  PROC DrawPart25()
    MoveL Offs(pOrigin,198.50,118.14,0.00),v40,z0,tPen\WObj:=wPaper;
    MoveL Offs(pOrigin,175.10,118.14,0.00),v40,z0,tPen\WObj:=wPaper;
    MoveL Offs(pOrigin,174.22,118.63,0.00),v40,z0,tPen\WObj:=wPaper;
    MoveL Offs(pOrigin,188.97,133.37,0.00),v40,fine,tPen\WObj:=wPaper;
    MoveL Offs(pOrigin,188.97,133.37,6.00),v60,z5,tPen\WObj:=wPaper;
    MoveL Offs(pOrigin,188.05,134.17,6.00),vTravel,z5,tPen\WObj:=wPaper;
    MoveL Offs(pOrigin,188.05,134.17,0.00),v60,z0,tPen\WObj:=wPaper;
    MoveL Offs(pOrigin,199.82,122.39,0.00),v40,z0,tPen\WObj:=wPaper;
    MoveL Offs(pOrigin,199.21,122.71,0.00),v40,z0,tPen\WObj:=wPaper;
    MoveL Offs(pOrigin,174.18,97.67,0.00),v40,z0,tPen\WObj:=wPaper;
    MoveL Offs(pOrigin,174.95,98.07,0.00),v40,z0,tPen\WObj:=wPaper;
    MoveL Offs(pOrigin,198.65,98.07,0.00),v40,z0,tPen\WObj:=wPaper;
    MoveL Offs(pOrigin,199.39,97.50,0.00),v40,z0,tPen\WObj:=wPaper;
    MoveL Offs(pOrigin,195.04,93.15,0.00),v40,z0,tPen\WObj:=wPaper;
    MoveL Offs(pOrigin,195.48,92.38,0.00),v40,z0,tPen\WObj:=wPaper;
    MoveL Offs(pOrigin,173.52,114.34,0.00),v40,z0,tPen\WObj:=wPaper;
    MoveL Offs(pOrigin,174.24,114.16,0.00),v40,z0,tPen\WObj:=wPaper;
    MoveL Offs(pOrigin,193.43,133.36,0.00),v40,z0,tPen\WObj:=wPaper;
    MoveL Offs(pOrigin,194.00,134.18,0.00),v40,z0,tPen\WObj:=wPaper;
    MoveL Offs(pOrigin,200.15,128.03,0.00),v40,z0,tPen\WObj:=wPaper;
    MoveL Offs(pOrigin,199.41,127.39,0.00),v40,z0,tPen\WObj:=wPaper;
    MoveL Offs(pOrigin,174.16,102.14,0.00),v40,z0,tPen\WObj:=wPaper;
    MoveL Offs(pOrigin,174.95,102.30,0.00),v40,z0,tPen\WObj:=wPaper;
    MoveL Offs(pOrigin,198.50,102.30,0.00),v40,z0,tPen\WObj:=wPaper;
    MoveL Offs(pOrigin,199.16,101.75,0.00),v40,z0,tPen\WObj:=wPaper;
    MoveL Offs(pOrigin,190.57,93.16,0.00),v40,z0,tPen\WObj:=wPaper;
    MoveL Offs(pOrigin,191.12,92.27,0.00),v40,z0,tPen\WObj:=wPaper;
    MoveL Offs(pOrigin,173.40,109.98,0.00),v40,z0,tPen\WObj:=wPaper;
    MoveL Offs(pOrigin,174.25,109.69,0.00),v40,z0,tPen\WObj:=wPaper;
    MoveL Offs(pOrigin,197.90,133.35,0.00),v40,z0,tPen\WObj:=wPaper;
    MoveL Offs(pOrigin,197.19,133.98,0.00),v40,z0,tPen\WObj:=wPaper;
    MoveL Offs(pOrigin,224.03,107.14,0.00),v40,z0,tPen\WObj:=wPaper;
    MoveL Offs(pOrigin,223.28,106.40,0.00),v40,z0,tPen\WObj:=wPaper;
    MoveL Offs(pOrigin,201.11,128.57,0.00),v40,z0,tPen\WObj:=wPaper;
    MoveL Offs(pOrigin,201.85,128.34,0.00),v40,z0,tPen\WObj:=wPaper;
    MoveL Offs(pOrigin,206.84,133.32,0.00),v40,z0,tPen\WObj:=wPaper;
    MoveL Offs(pOrigin,207.40,134.22,0.00),v40,z0,tPen\WObj:=wPaper;
    MoveL Offs(pOrigin,225.97,115.66,0.00),v40,z0,tPen\WObj:=wPaper;
    MoveL Offs(pOrigin,224.97,115.61,0.00),v40,z0,tPen\WObj:=wPaper;
    MoveL Offs(pOrigin,202.80,93.45,0.00),v40,z0,tPen\WObj:=wPaper;
    MoveL Offs(pOrigin,202.85,92.93,0.00),v40,z0,tPen\WObj:=wPaper;
    MoveL Offs(pOrigin,218.60,92.93,0.00),v40,z0,tPen\WObj:=wPaper;
    MoveL Offs(pOrigin,202.85,92.93,0.00),v40,z0,tPen\WObj:=wPaper;
    MoveL Offs(pOrigin,202.71,92.62,0.00),v40,z0,tPen\WObj:=wPaper;
    MoveL Offs(pOrigin,201.55,93.78,0.00),v40,z0,tPen\WObj:=wPaper;
    MoveL Offs(pOrigin,201.95,93.53,0.00),v40,z0,tPen\WObj:=wPaper;
    MoveL Offs(pOrigin,201.95,94.72,0.00),v40,z0,tPen\WObj:=wPaper;
    MoveL Offs(pOrigin,201.95,93.53,0.00),v40,z0,tPen\WObj:=wPaper;
    MoveL Offs(pOrigin,202.16,94.30,0.00),v40,z0,tPen\WObj:=wPaper;
    MoveL Offs(pOrigin,224.97,117.10,0.00),v40,z0,tPen\WObj:=wPaper;
    MoveL Offs(pOrigin,224.15,117.08,0.00),v40,z0,tPen\WObj:=wPaper;
    MoveL Offs(pOrigin,203.00,117.08,0.00),v40,z0,tPen\WObj:=wPaper;
    MoveL Offs(pOrigin,202.20,116.74,0.00),v40,z0,tPen\WObj:=wPaper;
    MoveL Offs(pOrigin,216.31,130.85,0.00),v40,z0,tPen\WObj:=wPaper;
    MoveL Offs(pOrigin,217.10,130.48,0.00),v40,z0,tPen\WObj:=wPaper;
    MoveL Offs(pOrigin,219.35,128.77,0.00),v40,z0,tPen\WObj:=wPaper;
    MoveL Offs(pOrigin,220.70,127.43,0.00),v40,z0,tPen\WObj:=wPaper;
    MoveL Offs(pOrigin,223.00,124.12,0.00),v40,z0,tPen\WObj:=wPaper;
    MoveL Offs(pOrigin,224.20,121.43,0.00),v40,z0,tPen\WObj:=wPaper;
    MoveL Offs(pOrigin,225.05,118.12,0.00),v40,z0,tPen\WObj:=wPaper;
    MoveL Offs(pOrigin,225.05,113.03,0.00),v40,z0,tPen\WObj:=wPaper;
    MoveL Offs(pOrigin,223.90,108.97,0.00),v40,z0,tPen\WObj:=wPaper;
    MoveL Offs(pOrigin,222.70,106.57,0.00),v40,z0,tPen\WObj:=wPaper;
    MoveL Offs(pOrigin,220.55,103.72,0.00),v40,z0,tPen\WObj:=wPaper;
    MoveL Offs(pOrigin,217.75,101.32,0.00),v40,z0,tPen\WObj:=wPaper;
    MoveL Offs(pOrigin,220.60,99.28,0.00),v40,z0,tPen\WObj:=wPaper;
    MoveL Offs(pOrigin,201.95,106.28,0.00),v40,z0,tPen\WObj:=wPaper;
    MoveL Offs(pOrigin,202.00,133.07,0.00),v40,z0,tPen\WObj:=wPaper;
    MoveL Offs(pOrigin,208.55,133.27,0.00),v40,z0,tPen\WObj:=wPaper;
    MoveL Offs(pOrigin,213.80,132.12,0.00),v40,z0,tPen\WObj:=wPaper;
    MoveL Offs(pOrigin,217.10,130.48,0.00),v40,z0,tPen\WObj:=wPaper;
    MoveL Offs(pOrigin,217.27,130.31,0.00),v40,z0,tPen\WObj:=wPaper;
    MoveL Offs(pOrigin,202.21,115.25,0.00),v40,z0,tPen\WObj:=wPaper;
    MoveL Offs(pOrigin,201.50,114.74,0.00),v40,z0,tPen\WObj:=wPaper;
    MoveL Offs(pOrigin,224.20,92.04,0.00),v40,z0,tPen\WObj:=wPaper;
    MoveL Offs(pOrigin,224.71,92.96,0.00),v40,z0,tPen\WObj:=wPaper;
    MoveL Offs(pOrigin,226.20,94.44,0.00),v40,z0,tPen\WObj:=wPaper;
    MoveL Offs(pOrigin,225.45,95.19,0.00),v40,z0,tPen\WObj:=wPaper;
    MoveL Offs(pOrigin,223.23,92.96,0.00),v40,z0,tPen\WObj:=wPaper;
    MoveL Offs(pOrigin,222.71,92.04,0.00),v40,z0,tPen\WObj:=wPaper;
    MoveL Offs(pOrigin,201.49,113.25,0.00),v40,z0,tPen\WObj:=wPaper;
    MoveL Offs(pOrigin,202.21,113.76,0.00),v40,z0,tPen\WObj:=wPaper;
    MoveL Offs(pOrigin,218.12,129.67,0.00),v40,z0,tPen\WObj:=wPaper;
    MoveL Offs(pOrigin,218.56,130.53,0.00),v40,z0,tPen\WObj:=wPaper;
    MoveL Offs(pOrigin,219.62,129.47,0.00),v40,z0,tPen\WObj:=wPaper;
    MoveL Offs(pOrigin,218.97,129.03,0.00),v40,z0,tPen\WObj:=wPaper;
    MoveL Offs(pOrigin,202.22,112.27,0.00),v40,z0,tPen\WObj:=wPaper;
    MoveL Offs(pOrigin,203.00,111.80,0.00),v40,z0,tPen\WObj:=wPaper;
    MoveL Offs(pOrigin,223.85,111.80,0.00),v40,z0,tPen\WObj:=wPaper;
    MoveL Offs(pOrigin,224.00,112.86,0.00),v40,z0,tPen\WObj:=wPaper;
    MoveL Offs(pOrigin,203.00,112.86,0.00),v40,z0,tPen\WObj:=wPaper;
    MoveL Offs(pOrigin,203.15,113.91,0.00),v40,z0,tPen\WObj:=wPaper;
    MoveL Offs(pOrigin,224.00,113.91,0.00),v40,z0,tPen\WObj:=wPaper;
    MoveL Offs(pOrigin,224.97,114.12,0.00),v40,z0,tPen\WObj:=wPaper;
    MoveL Offs(pOrigin,203.97,93.12,0.00),v40,z0,tPen\WObj:=wPaper;
    MoveL Offs(pOrigin,204.41,92.41,0.00),v40,z0,tPen\WObj:=wPaper;
    MoveL Offs(pOrigin,201.44,95.38,0.00),v40,z0,tPen\WObj:=wPaper;
    MoveL Offs(pOrigin,202.05,95.68,0.00),v40,z0,tPen\WObj:=wPaper;
    MoveL Offs(pOrigin,224.75,118.38,0.00),v40,z0,tPen\WObj:=wPaper;
    MoveL Offs(pOrigin,224.00,118.14,0.00),v40,z0,tPen\WObj:=wPaper;
    MoveL Offs(pOrigin,203.00,118.14,0.00),v40,z0,tPen\WObj:=wPaper;
    MoveL Offs(pOrigin,202.09,118.12,0.00),v40,z0,tPen\WObj:=wPaper;
    MoveL Offs(pOrigin,215.35,131.38,0.00),v40,z0,tPen\WObj:=wPaper;
    MoveL Offs(pOrigin,214.70,130.81,0.00),v40,z0,tPen\WObj:=wPaper;
    MoveL Offs(pOrigin,202.70,130.81,0.00),v40,z0,tPen\WObj:=wPaper;
    MoveL Offs(pOrigin,201.74,131.21,0.00),v40,z0,tPen\WObj:=wPaper;
    MoveL Offs(pOrigin,203.86,133.33,0.00),v40,z0,tPen\WObj:=wPaper;
    MoveL Offs(pOrigin,203.15,134.00,0.00),v40,z0,tPen\WObj:=wPaper;
    MoveL Offs(pOrigin,225.32,111.83,0.00),v40,z0,tPen\WObj:=wPaper;
    MoveL Offs(pOrigin,224.77,112.42,0.00),v40,z0,tPen\WObj:=wPaper;
    MoveL Offs(pOrigin,205.46,93.12,0.00),v40,z0,tPen\WObj:=wPaper;
    MoveL Offs(pOrigin,205.90,92.41,0.00),v40,z0,tPen\WObj:=wPaper;
    MoveL Offs(pOrigin,201.34,96.97,0.00),v40,z0,tPen\WObj:=wPaper;
    MoveL Offs(pOrigin,201.95,96.68,0.00),v40,z0,tPen\WObj:=wPaper;
    MoveL Offs(pOrigin,201.95,105.82,0.00),v40,z0,tPen\WObj:=wPaper;
    MoveL Offs(pOrigin,201.95,96.68,0.00),v40,z0,tPen\WObj:=wPaper;
    MoveL Offs(pOrigin,202.05,97.17,0.00),v40,z0,tPen\WObj:=wPaper;
    MoveL Offs(pOrigin,224.53,119.66,0.00),v40,z0,tPen\WObj:=wPaper;
    MoveL Offs(pOrigin,223.85,119.19,0.00),v40,z0,tPen\WObj:=wPaper;
    MoveL Offs(pOrigin,203.00,119.19,0.00),v40,z0,tPen\WObj:=wPaper;
  ENDPROC

  PROC DrawPart26()
    MoveL Offs(pOrigin,202.09,119.61,0.00),v40,z0,tPen\WObj:=wPaper;
    MoveL Offs(pOrigin,214.39,131.92,0.00),v40,z0,tPen\WObj:=wPaper;
    MoveL Offs(pOrigin,214.74,132.86,0.00),v40,z0,tPen\WObj:=wPaper;
    MoveL Offs(pOrigin,224.71,122.89,0.00),v40,z0,tPen\WObj:=wPaper;
    MoveL Offs(pOrigin,223.99,122.10,0.00),v40,z0,tPen\WObj:=wPaper;
    MoveL Offs(pOrigin,202.04,100.15,0.00),v40,z0,tPen\WObj:=wPaper;
    MoveL Offs(pOrigin,201.46,99.85,0.00),v40,z0,tPen\WObj:=wPaper;
    MoveL Offs(pOrigin,208.88,92.42,0.00),v40,z0,tPen\WObj:=wPaper;
    MoveL Offs(pOrigin,208.44,93.11,0.00),v40,z0,tPen\WObj:=wPaper;
    MoveL Offs(pOrigin,223.40,108.07,0.00),v40,z0,tPen\WObj:=wPaper;
    MoveL Offs(pOrigin,222.80,108.63,0.00),v40,z0,tPen\WObj:=wPaper;
    MoveL Offs(pOrigin,203.15,108.63,0.00),v40,z0,tPen\WObj:=wPaper;
    MoveL Offs(pOrigin,203.15,109.69,0.00),v40,z0,tPen\WObj:=wPaper;
    MoveL Offs(pOrigin,223.25,109.69,0.00),v40,z0,tPen\WObj:=wPaper;
    MoveL Offs(pOrigin,223.55,110.74,0.00),v40,z0,tPen\WObj:=wPaper;
    MoveL Offs(pOrigin,203.00,110.74,0.00),v40,z0,tPen\WObj:=wPaper;
    MoveL Offs(pOrigin,202.11,110.68,0.00),v40,z0,tPen\WObj:=wPaper;
    MoveL Offs(pOrigin,219.72,128.29,0.00),v40,z0,tPen\WObj:=wPaper;
    MoveL Offs(pOrigin,219.95,128.02,0.00),v40,z0,tPen\WObj:=wPaper;
    MoveL Offs(pOrigin,219.50,128.48,0.00),v40,z0,tPen\WObj:=wPaper;
    MoveL Offs(pOrigin,219.95,128.02,0.00),v40,z0,tPen\WObj:=wPaper;
    MoveL Offs(pOrigin,220.47,127.54,0.00),v40,z0,tPen\WObj:=wPaper;
    MoveL Offs(pOrigin,202.12,109.19,0.00),v40,z0,tPen\WObj:=wPaper;
    MoveL Offs(pOrigin,201.48,108.78,0.00),v40,z0,tPen\WObj:=wPaper;
    MoveL Offs(pOrigin,218.03,92.24,0.00),v40,z0,tPen\WObj:=wPaper;
    MoveL Offs(pOrigin,217.38,93.08,0.00),v40,z0,tPen\WObj:=wPaper;
    MoveL Offs(pOrigin,222.36,98.07,0.00),v40,z0,tPen\WObj:=wPaper;
    MoveL Offs(pOrigin,223.11,97.32,0.00),v40,z0,tPen\WObj:=wPaper;
    MoveL Offs(pOrigin,218.86,93.08,0.00),v40,z0,tPen\WObj:=wPaper;
    MoveL Offs(pOrigin,219.05,92.93,0.00),v40,z0,tPen\WObj:=wPaper;
    MoveL Offs(pOrigin,227.10,93.07,0.00),v40,z0,tPen\WObj:=wPaper;
    MoveL Offs(pOrigin,227.10,93.53,0.00),v40,z0,tPen\WObj:=wPaper;
    MoveL Offs(pOrigin,223.40,97.22,0.00),v40,z0,tPen\WObj:=wPaper;
    MoveL Offs(pOrigin,220.90,99.12,0.00),v40,z0,tPen\WObj:=wPaper;
    MoveL Offs(pOrigin,219.05,92.93,0.00),v40,z0,tPen\WObj:=wPaper;
    MoveL Offs(pOrigin,220.14,92.86,0.00),v40,z0,tPen\WObj:=wPaper;
    MoveL Offs(pOrigin,223.85,96.58,0.00),v40,z0,tPen\WObj:=wPaper;
    MoveL Offs(pOrigin,223.40,95.96,0.00),v40,z0,tPen\WObj:=wPaper;
    MoveL Offs(pOrigin,202.85,95.96,0.00),v40,z0,tPen\WObj:=wPaper;
    MoveL Offs(pOrigin,202.85,94.90,0.00),v40,z0,tPen\WObj:=wPaper;
    MoveL Offs(pOrigin,224.60,94.90,0.00),v40,z0,tPen\WObj:=wPaper;
    MoveL Offs(pOrigin,224.71,95.94,0.00),v40,z0,tPen\WObj:=wPaper;
    MoveL Offs(pOrigin,221.74,92.97,0.00),v40,fine,tPen\WObj:=wPaper;
    MoveL Offs(pOrigin,221.74,92.97,6.00),v60,z5,tPen\WObj:=wPaper;
    MoveL Offs(pOrigin,222.38,90.62,6.00),vTravel,z5,tPen\WObj:=wPaper;
    MoveL Offs(pOrigin,222.38,90.62,0.00),v60,z0,tPen\WObj:=wPaper;
    MoveL Offs(pOrigin,202.12,70.37,0.00),v40,z0,tPen\WObj:=wPaper;
    MoveL Offs(pOrigin,201.37,70.06,0.00),v40,z0,tPen\WObj:=wPaper;
    MoveL Offs(pOrigin,218.66,52.78,0.00),v40,z0,tPen\WObj:=wPaper;
    MoveL Offs(pOrigin,217.91,53.30,0.00),v40,z0,tPen\WObj:=wPaper;
    MoveL Offs(pOrigin,229.58,64.97,0.00),v40,z0,tPen\WObj:=wPaper;
    MoveL Offs(pOrigin,228.80,65.34,0.00),v40,z0,tPen\WObj:=wPaper;
    MoveL Offs(pOrigin,203.15,65.34,0.00),v40,z0,tPen\WObj:=wPaper;
    MoveL Offs(pOrigin,203.15,64.28,0.00),v40,z0,tPen\WObj:=wPaper;
    MoveL Offs(pOrigin,228.20,64.28,0.00),v40,fine,tPen\WObj:=wPaper;
    MoveL Offs(pOrigin,228.20,64.28,6.00),v60,z5,tPen\WObj:=wPaper;
    MoveL Offs(pOrigin,227.60,63.22,6.00),vTravel,z5,tPen\WObj:=wPaper;
    MoveL Offs(pOrigin,227.60,63.22,0.00),v60,z0,tPen\WObj:=wPaper;
    MoveL Offs(pOrigin,203.00,63.22,0.00),v40,z0,tPen\WObj:=wPaper;
    MoveL Offs(pOrigin,202.14,62.92,0.00),v40,z0,tPen\WObj:=wPaper;
    MoveL Offs(pOrigin,229.19,89.97,0.00),v40,z0,tPen\WObj:=wPaper;
    MoveL Offs(pOrigin,229.10,90.38,0.00),v40,z0,tPen\WObj:=wPaper;
    MoveL Offs(pOrigin,230.55,87.68,0.00),v40,z0,tPen\WObj:=wPaper;
    MoveL Offs(pOrigin,231.80,83.78,0.00),v40,z0,tPen\WObj:=wPaper;
    MoveL Offs(pOrigin,232.40,79.28,0.00),v40,z0,tPen\WObj:=wPaper;
    MoveL Offs(pOrigin,232.40,75.82,0.00),v40,z0,tPen\WObj:=wPaper;
    MoveL Offs(pOrigin,231.80,71.18,0.00),v40,z0,tPen\WObj:=wPaper;
    MoveL Offs(pOrigin,230.50,66.97,0.00),v40,z0,tPen\WObj:=wPaper;
    MoveL Offs(pOrigin,227.45,61.42,0.00),v40,z0,tPen\WObj:=wPaper;
    MoveL Offs(pOrigin,225.80,59.33,0.00),v40,z0,tPen\WObj:=wPaper;
    MoveL Offs(pOrigin,222.65,56.33,0.00),v40,z0,tPen\WObj:=wPaper;
    MoveL Offs(pOrigin,218.90,53.88,0.00),v40,z0,tPen\WObj:=wPaper;
    MoveL Offs(pOrigin,215.30,52.22,0.00),v40,z0,tPen\WObj:=wPaper;
    MoveL Offs(pOrigin,209.00,50.78,0.00),v40,z0,tPen\WObj:=wPaper;
    MoveL Offs(pOrigin,201.95,50.83,0.00),v40,z0,tPen\WObj:=wPaper;
    MoveL Offs(pOrigin,202.00,90.47,0.00),v40,z0,tPen\WObj:=wPaper;
    MoveL Offs(pOrigin,229.10,90.38,0.00),v40,z0,tPen\WObj:=wPaper;
    MoveL Offs(pOrigin,228.34,90.61,0.00),v40,z0,tPen\WObj:=wPaper;
    MoveL Offs(pOrigin,202.14,64.41,0.00),v40,z0,tPen\WObj:=wPaper;
    MoveL Offs(pOrigin,201.46,64.00,0.00),v40,z0,tPen\WObj:=wPaper;
    MoveL Offs(pOrigin,214.29,51.17,0.00),v40,z0,tPen\WObj:=wPaper;
    MoveL Offs(pOrigin,213.24,51.61,0.00),v40,z0,tPen\WObj:=wPaper;
    MoveL Offs(pOrigin,231.38,69.75,0.00),v40,z0,tPen\WObj:=wPaper;
    MoveL Offs(pOrigin,232.00,69.30,0.00),v40,z0,tPen\WObj:=wPaper;
    MoveL Offs(pOrigin,210.37,90.94,0.00),v40,z0,tPen\WObj:=wPaper;
    MoveL Offs(pOrigin,210.04,90.23,0.00),v40,z0,tPen\WObj:=wPaper;
    MoveL Offs(pOrigin,202.19,82.38,0.00),v40,z0,tPen\WObj:=wPaper;
    MoveL Offs(pOrigin,201.51,81.87,0.00),v40,z0,tPen\WObj:=wPaper;
    MoveL Offs(pOrigin,225.48,57.90,0.00),v40,z0,tPen\WObj:=wPaper;
    MoveL Offs(pOrigin,226.23,58.65,0.00),v40,z0,tPen\WObj:=wPaper;
    MoveL Offs(pOrigin,201.41,83.47,0.00),v40,z0,tPen\WObj:=wPaper;
    MoveL Offs(pOrigin,202.19,83.87,0.00),v40,z0,tPen\WObj:=wPaper;
    MoveL Offs(pOrigin,208.77,90.45,0.00),v40,z0,tPen\WObj:=wPaper;
    MoveL Offs(pOrigin,208.88,90.93,0.00),v40,z0,tPen\WObj:=wPaper;
    MoveL Offs(pOrigin,231.79,68.02,0.00),v40,z0,tPen\WObj:=wPaper;
    MoveL Offs(pOrigin,230.74,67.62,0.00),v40,z0,tPen\WObj:=wPaper;
    MoveL Offs(pOrigin,215.58,52.46,0.00),v40,z0,tPen\WObj:=wPaper;
    MoveL Offs(pOrigin,215.47,51.49,0.00),v40,z0,tPen\WObj:=wPaper;
    MoveL Offs(pOrigin,201.57,65.38,0.00),v40,z0,tPen\WObj:=wPaper;
    MoveL Offs(pOrigin,202.14,65.90,0.00),v40,z0,tPen\WObj:=wPaper;
    MoveL Offs(pOrigin,226.85,90.61,0.00),v40,fine,tPen\WObj:=wPaper;
    MoveL Offs(pOrigin,226.85,90.61,6.00),v60,z5,tPen\WObj:=wPaper;
    MoveL Offs(pOrigin,227.71,91.52,6.00),vTravel,z5,tPen\WObj:=wPaper;
    MoveL Offs(pOrigin,227.71,91.52,0.00),v60,z0,tPen\WObj:=wPaper;
    MoveL Offs(pOrigin,231.95,87.28,0.00),v40,z0,tPen\WObj:=wPaper;
    MoveL Offs(pOrigin,230.90,87.20,0.00),v40,z0,tPen\WObj:=wPaper;
    MoveL Offs(pOrigin,202.05,58.35,0.00),v40,z0,tPen\WObj:=wPaper;
    MoveL Offs(pOrigin,201.44,58.04,0.00),v40,z0,tPen\WObj:=wPaper;
    MoveL Offs(pOrigin,209.50,49.98,0.00),v40,z0,tPen\WObj:=wPaper;
    MoveL Offs(pOrigin,209.52,50.88,0.00),v40,z0,tPen\WObj:=wPaper;
    MoveL Offs(pOrigin,232.11,73.47,0.00),v40,z0,tPen\WObj:=wPaper;
    MoveL Offs(pOrigin,231.20,73.78,0.00),v40,z0,tPen\WObj:=wPaper;
    MoveL Offs(pOrigin,203.15,73.78,0.00),v40,z0,tPen\WObj:=wPaper;
    MoveL Offs(pOrigin,202.33,73.56,0.00),v40,z0,tPen\WObj:=wPaper;
    MoveL Offs(pOrigin,219.30,90.53,0.00),v40,z0,tPen\WObj:=wPaper;
    MoveL Offs(pOrigin,219.20,91.07,0.00),v40,z0,tPen\WObj:=wPaper;
    MoveL Offs(pOrigin,233.41,76.86,0.00),v40,z0,tPen\WObj:=wPaper;
    MoveL Offs(pOrigin,232.42,76.77,0.00),v40,z0,tPen\WObj:=wPaper;
    MoveL Offs(pOrigin,206.33,50.67,0.00),v40,fine,tPen\WObj:=wPaper;
    MoveL Offs(pOrigin,206.33,50.67,6.00),v60,z5,tPen\WObj:=wPaper;
  ENDPROC

  PROC DrawPart27()
    MoveL Offs(pOrigin,206.95,49.55,6.00),vTravel,z5,tPen\WObj:=wPaper;
    MoveL Offs(pOrigin,206.95,49.55,0.00),v60,z0,tPen\WObj:=wPaper;
    MoveL Offs(pOrigin,201.01,55.49,0.00),v40,z0,tPen\WObj:=wPaper;
    MoveL Offs(pOrigin,201.85,55.16,0.00),v40,z0,tPen\WObj:=wPaper;
    MoveL Offs(pOrigin,231.44,84.75,0.00),v40,z0,tPen\WObj:=wPaper;
    MoveL Offs(pOrigin,230.60,84.34,0.00),v40,z0,tPen\WObj:=wPaper;
    MoveL Offs(pOrigin,203.00,84.34,0.00),v40,z0,tPen\WObj:=wPaper;
    MoveL Offs(pOrigin,203.00,85.40,0.00),v40,z0,tPen\WObj:=wPaper;
    MoveL Offs(pOrigin,230.45,85.40,0.00),v40,z0,tPen\WObj:=wPaper;
    MoveL Offs(pOrigin,231.12,85.92,0.00),v40,z0,tPen\WObj:=wPaper;
    MoveL Offs(pOrigin,202.05,56.86,0.00),v40,z0,tPen\WObj:=wPaper;
    MoveL Offs(pOrigin,202.85,56.89,0.00),v40,z0,tPen\WObj:=wPaper;
    MoveL Offs(pOrigin,221.75,56.89,0.00),v40,fine,tPen\WObj:=wPaper;
    MoveL Offs(pOrigin,221.75,56.89,6.00),v60,z5,tPen\WObj:=wPaper;
    MoveL Offs(pOrigin,223.22,57.12,6.00),vTravel,z5,tPen\WObj:=wPaper;
    MoveL Offs(pOrigin,223.22,57.12,0.00),v60,z0,tPen\WObj:=wPaper;
    MoveL Offs(pOrigin,226.51,60.40,0.00),v40,z0,tPen\WObj:=wPaper;
    MoveL Offs(pOrigin,226.10,61.11,0.00),v40,z0,tPen\WObj:=wPaper;
    MoveL Offs(pOrigin,203.00,61.11,0.00),v40,z0,tPen\WObj:=wPaper;
    MoveL Offs(pOrigin,202.04,61.32,0.00),v40,z0,tPen\WObj:=wPaper;
    MoveL Offs(pOrigin,229.83,89.11,0.00),v40,z0,tPen\WObj:=wPaper;
    MoveL Offs(pOrigin,229.10,88.57,0.00),v40,z0,tPen\WObj:=wPaper;
    MoveL Offs(pOrigin,203.15,88.57,0.00),v40,z0,tPen\WObj:=wPaper;
    MoveL Offs(pOrigin,202.18,88.34,0.00),v40,z0,tPen\WObj:=wPaper;
    MoveL Offs(pOrigin,204.09,90.25,0.00),v40,z0,tPen\WObj:=wPaper;
    MoveL Offs(pOrigin,204.52,90.81,0.00),v40,z0,tPen\WObj:=wPaper;
    MoveL Offs(pOrigin,230.61,64.72,0.00),v40,z0,tPen\WObj:=wPaper;
    MoveL Offs(pOrigin,229.97,63.87,0.00),v40,z0,tPen\WObj:=wPaper;
    MoveL Offs(pOrigin,203.13,90.70,0.00),v40,z0,tPen\WObj:=wPaper;
    MoveL Offs(pOrigin,202.07,90.28,0.00),v40,z0,tPen\WObj:=wPaper;
    MoveL Offs(pOrigin,229.43,62.91,0.00),v40,z0,tPen\WObj:=wPaper;
    MoveL Offs(pOrigin,228.90,61.95,0.00),v40,z0,tPen\WObj:=wPaper;
    MoveL Offs(pOrigin,201.53,89.32,0.00),v40,fine,tPen\WObj:=wPaper;
    MoveL Offs(pOrigin,201.53,89.32,6.00),v60,z5,tPen\WObj:=wPaper;
    MoveL Offs(pOrigin,201.53,87.83,6.00),vTravel,z5,tPen\WObj:=wPaper;
    MoveL Offs(pOrigin,201.53,87.83,0.00),v60,z0,tPen\WObj:=wPaper;
    MoveL Offs(pOrigin,228.26,61.10,0.00),v40,z0,tPen\WObj:=wPaper;
    MoveL Offs(pOrigin,227.45,61.58,0.00),v40,z0,tPen\WObj:=wPaper;
    MoveL Offs(pOrigin,227.75,62.03,0.00),v40,z0,tPen\WObj:=wPaper;
    MoveL Offs(pOrigin,227.45,61.58,0.00),v40,z0,tPen\WObj:=wPaper;
    MoveL Offs(pOrigin,226.85,62.17,0.00),v40,z0,tPen\WObj:=wPaper;
    MoveL Offs(pOrigin,203.00,62.17,0.00),v40,fine,tPen\WObj:=wPaper;
    MoveL Offs(pOrigin,203.00,62.17,6.00),v60,z5,tPen\WObj:=wPaper;
    MoveL Offs(pOrigin,201.46,62.51,6.00),vTravel,z5,tPen\WObj:=wPaper;
    MoveL Offs(pOrigin,201.46,62.51,0.00),v60,z0,tPen\WObj:=wPaper;
    MoveL Offs(pOrigin,213.23,50.74,0.00),v40,fine,tPen\WObj:=wPaper;
    MoveL Offs(pOrigin,213.23,50.74,6.00),v60,z5,tPen\WObj:=wPaper;
    MoveL Offs(pOrigin,212.06,50.42,6.00),vTravel,z5,tPen\WObj:=wPaper;
    MoveL Offs(pOrigin,212.06,50.42,0.00),v60,z0,tPen\WObj:=wPaper;
    MoveL Offs(pOrigin,201.45,61.02,0.00),v40,fine,tPen\WObj:=wPaper;
    MoveL Offs(pOrigin,201.45,61.02,6.00),v60,z5,tPen\WObj:=wPaper;
    MoveL Offs(pOrigin,202.15,59.94,6.00),vTravel,z5,tPen\WObj:=wPaper;
    MoveL Offs(pOrigin,202.15,59.94,0.00),v60,z0,tPen\WObj:=wPaper;
    MoveL Offs(pOrigin,230.26,88.05,0.00),v40,z0,tPen\WObj:=wPaper;
    MoveL Offs(pOrigin,229.70,87.51,0.00),v40,z0,tPen\WObj:=wPaper;
    MoveL Offs(pOrigin,203.00,87.51,0.00),v40,z0,tPen\WObj:=wPaper;
    MoveL Offs(pOrigin,202.18,86.85,0.00),v40,z0,tPen\WObj:=wPaper;
    MoveL Offs(pOrigin,205.79,90.46,0.00),v40,z0,tPen\WObj:=wPaper;
    MoveL Offs(pOrigin,205.90,90.92,0.00),v40,z0,tPen\WObj:=wPaper;
    MoveL Offs(pOrigin,231.14,65.68,0.00),v40,z0,tPen\WObj:=wPaper;
    MoveL Offs(pOrigin,231.68,66.64,0.00),v40,z0,tPen\WObj:=wPaper;
    MoveL Offs(pOrigin,207.18,91.14,0.00),v40,z0,tPen\WObj:=wPaper;
    MoveL Offs(pOrigin,207.28,90.45,0.00),v40,z0,tPen\WObj:=wPaper;
    MoveL Offs(pOrigin,202.19,85.36,0.00),v40,z0,tPen\WObj:=wPaper;
    MoveL Offs(pOrigin,201.41,84.96,0.00),v40,z0,tPen\WObj:=wPaper;
    MoveL Offs(pOrigin,226.76,59.61,0.00),v40,z0,tPen\WObj:=wPaper;
    MoveL Offs(pOrigin,225.95,59.78,0.00),v40,z0,tPen\WObj:=wPaper;
    MoveL Offs(pOrigin,226.70,60.53,0.00),v40,z0,tPen\WObj:=wPaper;
    MoveL Offs(pOrigin,225.95,59.78,0.00),v40,z0,tPen\WObj:=wPaper;
    MoveL Offs(pOrigin,225.20,60.06,0.00),v40,z0,tPen\WObj:=wPaper;
    MoveL Offs(pOrigin,203.00,60.06,0.00),v40,z0,tPen\WObj:=wPaper;
    MoveL Offs(pOrigin,203.00,59.00,0.00),v40,z0,tPen\WObj:=wPaper;
    MoveL Offs(pOrigin,224.15,59.00,0.00),v40,fine,tPen\WObj:=wPaper;
    MoveL Offs(pOrigin,224.15,59.00,6.00),v60,z5,tPen\WObj:=wPaper;
    MoveL Offs(pOrigin,222.95,57.94,6.00),vTravel,z5,tPen\WObj:=wPaper;
    MoveL Offs(pOrigin,222.95,57.94,0.00),v60,z0,tPen\WObj:=wPaper;
    MoveL Offs(pOrigin,203.00,57.94,0.00),v40,fine,tPen\WObj:=wPaper;
    MoveL Offs(pOrigin,203.00,57.94,6.00),v60,z5,tPen\WObj:=wPaper;
    MoveL Offs(pOrigin,202.85,55.83,6.00),vTravel,z5,tPen\WObj:=wPaper;
    MoveL Offs(pOrigin,202.85,55.83,0.00),v60,z0,tPen\WObj:=wPaper;
    MoveL Offs(pOrigin,220.40,55.83,0.00),v40,fine,tPen\WObj:=wPaper;
    MoveL Offs(pOrigin,220.40,55.83,6.00),v60,z5,tPen\WObj:=wPaper;
    MoveL Offs(pOrigin,219.80,54.53,6.00),vTravel,z5,tPen\WObj:=wPaper;
    MoveL Offs(pOrigin,219.80,54.53,0.00),v60,z0,tPen\WObj:=wPaper;
    MoveL Offs(pOrigin,220.25,54.83,0.00),v40,z0,tPen\WObj:=wPaper;
    MoveL Offs(pOrigin,219.80,54.53,0.00),v40,z0,tPen\WObj:=wPaper;
    MoveL Offs(pOrigin,220.58,53.84,0.00),v40,z0,tPen\WObj:=wPaper;
    MoveL Offs(pOrigin,201.49,72.94,0.00),v40,fine,tPen\WObj:=wPaper;
    MoveL Offs(pOrigin,201.49,72.94,6.00),v60,z5,tPen\WObj:=wPaper;
    MoveL Offs(pOrigin,202.33,72.07,6.00),vTravel,z5,tPen\WObj:=wPaper;
    MoveL Offs(pOrigin,202.33,72.07,0.00),v60,z0,tPen\WObj:=wPaper;
    MoveL Offs(pOrigin,220.89,90.63,0.00),v40,fine,tPen\WObj:=wPaper;
    MoveL Offs(pOrigin,220.89,90.63,6.00),v60,z5,tPen\WObj:=wPaper;
    MoveL Offs(pOrigin,223.56,91.19,6.00),vTravel,z5,tPen\WObj:=wPaper;
    MoveL Offs(pOrigin,223.56,91.19,0.00),v60,z0,tPen\WObj:=wPaper;
    MoveL Offs(pOrigin,233.10,81.64,0.00),v40,z0,tPen\WObj:=wPaper;
    MoveL Offs(pOrigin,232.19,81.02,0.00),v40,z0,tPen\WObj:=wPaper;
    MoveL Offs(pOrigin,202.39,51.22,0.00),v40,z0,tPen\WObj:=wPaper;
    MoveL Offs(pOrigin,203.30,51.61,0.00),v40,z0,tPen\WObj:=wPaper;
    MoveL Offs(pOrigin,209.75,51.61,0.00),v40,fine,tPen\WObj:=wPaper;
    MoveL Offs(pOrigin,209.75,51.61,6.00),v60,z5,tPen\WObj:=wPaper;
    MoveL Offs(pOrigin,211.22,51.09,6.00),vTravel,z5,tPen\WObj:=wPaper;
    MoveL Offs(pOrigin,211.22,51.09,0.00),v60,z0,tPen\WObj:=wPaper;
    MoveL Offs(pOrigin,232.01,71.88,0.00),v40,z0,tPen\WObj:=wPaper;
    MoveL Offs(pOrigin,232.86,71.43,0.00),v40,z0,tPen\WObj:=wPaper;
    MoveL Offs(pOrigin,213.13,91.16,0.00),v40,z0,tPen\WObj:=wPaper;
    MoveL Offs(pOrigin,213.23,90.44,0.00),v40,z0,tPen\WObj:=wPaper;
    MoveL Offs(pOrigin,202.42,79.62,0.00),v40,z0,tPen\WObj:=wPaper;
    MoveL Offs(pOrigin,203.15,80.12,0.00),v40,z0,tPen\WObj:=wPaper;
    MoveL Offs(pOrigin,231.35,80.12,0.00),v40,z0,tPen\WObj:=wPaper;
    MoveL Offs(pOrigin,231.35,79.06,0.00),v40,z0,tPen\WObj:=wPaper;
    MoveL Offs(pOrigin,203.15,79.06,0.00),v40,z0,tPen\WObj:=wPaper;
    MoveL Offs(pOrigin,203.15,78.01,0.00),v40,z0,tPen\WObj:=wPaper;
    MoveL Offs(pOrigin,231.50,78.01,0.00),v40,z0,tPen\WObj:=wPaper;
    MoveL Offs(pOrigin,232.42,78.26,0.00),v40,z0,tPen\WObj:=wPaper;
    MoveL Offs(pOrigin,204.94,50.79,0.00),v40,z0,tPen\WObj:=wPaper;
    MoveL Offs(pOrigin,205.25,49.76,0.00),v40,z0,tPen\WObj:=wPaper;
    MoveL Offs(pOrigin,201.01,54.00,0.00),v40,z0,tPen\WObj:=wPaper;
    MoveL Offs(pOrigin,201.85,53.67,0.00),v40,z0,tPen\WObj:=wPaper;
    MoveL Offs(pOrigin,231.76,83.58,0.00),v40,z0,tPen\WObj:=wPaper;
  ENDPROC

  PROC DrawPart28()
    MoveL Offs(pOrigin,232.47,83.77,0.00),v40,z0,tPen\WObj:=wPaper;
    MoveL Offs(pOrigin,225.15,91.09,0.00),v40,z0,tPen\WObj:=wPaper;
    MoveL Offs(pOrigin,225.25,90.51,0.00),v40,z0,tPen\WObj:=wPaper;
    MoveL Offs(pOrigin,202.13,67.39,0.00),v40,z0,tPen\WObj:=wPaper;
    MoveL Offs(pOrigin,201.58,66.87,0.00),v40,z0,tPen\WObj:=wPaper;
    MoveL Offs(pOrigin,216.85,51.60,0.00),v40,z0,tPen\WObj:=wPaper;
    MoveL Offs(pOrigin,217.81,52.13,0.00),v40,z0,tPen\WObj:=wPaper;
    MoveL Offs(pOrigin,201.47,68.47,0.00),v40,z0,tPen\WObj:=wPaper;
    MoveL Offs(pOrigin,202.13,68.88,0.00),v40,z0,tPen\WObj:=wPaper;
    MoveL Offs(pOrigin,223.76,90.51,0.00),v40,fine,tPen\WObj:=wPaper;
    MoveL Offs(pOrigin,223.76,90.51,6.00),v60,z5,tPen\WObj:=wPaper;
    MoveL Offs(pOrigin,225.20,93.85,6.00),vTravel,z5,tPen\WObj:=wPaper;
    MoveL Offs(pOrigin,225.20,93.85,0.00),v60,z0,tPen\WObj:=wPaper;
    MoveL Offs(pOrigin,203.15,93.85,0.00),v40,fine,tPen\WObj:=wPaper;
    MoveL Offs(pOrigin,203.15,93.85,6.00),v60,z5,tPen\WObj:=wPaper;
    MoveL Offs(pOrigin,201.95,94.88,6.00),vTravel,z5,tPen\WObj:=wPaper;
    MoveL Offs(pOrigin,201.95,94.88,0.00),v60,z0,tPen\WObj:=wPaper;
    MoveL Offs(pOrigin,201.95,96.38,0.00),v40,z0,tPen\WObj:=wPaper;
    MoveL Offs(pOrigin,201.95,94.88,0.00),v40,fine,tPen\WObj:=wPaper;
    MoveL Offs(pOrigin,201.95,94.88,6.00),v60,z5,tPen\WObj:=wPaper;
    MoveL Offs(pOrigin,199.85,95.48,6.00),vTravel,z5,tPen\WObj:=wPaper;
    MoveL Offs(pOrigin,199.85,95.48,0.00),v60,z0,tPen\WObj:=wPaper;
    MoveL Offs(pOrigin,173.54,121.79,0.00),v40,z0,tPen\WObj:=wPaper;
    MoveL Offs(pOrigin,174.32,121.71,0.00),v40,z0,tPen\WObj:=wPaper;
    MoveL Offs(pOrigin,185.88,133.27,0.00),v40,z0,tPen\WObj:=wPaper;
    MoveL Offs(pOrigin,186.56,134.16,0.00),v40,z0,tPen\WObj:=wPaper;
    MoveL Offs(pOrigin,199.92,120.80,0.00),v40,z0,tPen\WObj:=wPaper;
    MoveL Offs(pOrigin,199.21,121.22,0.00),v40,z0,tPen\WObj:=wPaper;
    MoveL Offs(pOrigin,174.18,96.19,0.00),v40,z0,tPen\WObj:=wPaper;
    MoveL Offs(pOrigin,173.47,96.47,0.00),v40,z0,tPen\WObj:=wPaper;
    MoveL Offs(pOrigin,199.88,70.06,0.00),v40,z0,tPen\WObj:=wPaper;
    MoveL Offs(pOrigin,199.04,70.27,0.00),v40,z0,tPen\WObj:=wPaper;
    MoveL Offs(pOrigin,179.52,50.75,0.00),v40,fine,tPen\WObj:=wPaper;
    MoveL Offs(pOrigin,179.52,50.75,6.00),v60,z5,tPen\WObj:=wPaper;
    MoveL Offs(pOrigin,180.04,49.58,6.00),vTravel,z5,tPen\WObj:=wPaper;
    MoveL Offs(pOrigin,180.04,49.58,0.00),v60,z0,tPen\WObj:=wPaper;
    MoveL Offs(pOrigin,173.25,56.37,0.00),v40,z0,tPen\WObj:=wPaper;
    MoveL Offs(pOrigin,174.30,55.98,0.00),v40,z0,tPen\WObj:=wPaper;
    MoveL Offs(pOrigin,199.11,80.80,0.00),v40,z0,tPen\WObj:=wPaper;
    MoveL Offs(pOrigin,199.59,80.80,0.00),v40,z0,tPen\WObj:=wPaper;
    MoveL Offs(pOrigin,189.52,90.88,0.00),v40,z0,tPen\WObj:=wPaper;
    MoveL Offs(pOrigin,189.20,90.29,0.00),v40,z0,tPen\WObj:=wPaper;
    MoveL Offs(pOrigin,174.24,75.34,0.00),v40,z0,tPen\WObj:=wPaper;
    MoveL Offs(pOrigin,175.25,74.84,0.00),v40,z0,tPen\WObj:=wPaper;
    MoveL Offs(pOrigin,198.35,74.84,0.00),v40,z0,tPen\WObj:=wPaper;
    MoveL Offs(pOrigin,199.13,74.84,0.00),v40,z0,tPen\WObj:=wPaper;
    MoveL Offs(pOrigin,175.16,50.87,0.00),v40,z0,tPen\WObj:=wPaper;
    MoveL Offs(pOrigin,174.50,50.83,0.00),v40,z0,tPen\WObj:=wPaper;
    MoveL Offs(pOrigin,198.65,50.62,0.00),v40,z0,tPen\WObj:=wPaper;
    MoveL Offs(pOrigin,199.35,50.92,0.00),v40,z0,tPen\WObj:=wPaper;
    MoveL Offs(pOrigin,199.35,90.47,0.00),v40,z0,tPen\WObj:=wPaper;
    MoveL Offs(pOrigin,174.40,90.38,0.00),v40,z0,tPen\WObj:=wPaper;
    MoveL Offs(pOrigin,174.50,50.83,0.00),v40,z0,tPen\WObj:=wPaper;
    MoveL Offs(pOrigin,174.41,51.62,0.00),v40,z0,tPen\WObj:=wPaper;
    MoveL Offs(pOrigin,199.13,76.33,0.00),v40,z0,tPen\WObj:=wPaper;
    MoveL Offs(pOrigin,199.79,76.12,0.00),v40,z0,tPen\WObj:=wPaper;
    MoveL Offs(pOrigin,184.73,91.18,0.00),v40,z0,tPen\WObj:=wPaper;
    MoveL Offs(pOrigin,185.05,90.62,0.00),v40,z0,tPen\WObj:=wPaper;
    MoveL Offs(pOrigin,174.23,79.80,0.00),v40,z0,tPen\WObj:=wPaper;
    MoveL Offs(pOrigin,173.53,79.98,0.00),v40,z0,tPen\WObj:=wPaper;
    MoveL Offs(pOrigin,200.15,53.36,0.00),v40,z0,tPen\WObj:=wPaper;
    MoveL Offs(pOrigin,199.41,52.72,0.00),v40,z0,tPen\WObj:=wPaper;
    MoveL Offs(pOrigin,197.50,50.81,0.00),v40,z0,tPen\WObj:=wPaper;
    MoveL Offs(pOrigin,198.20,51.61,0.00),v40,z0,tPen\WObj:=wPaper;
    MoveL Offs(pOrigin,175.55,51.61,0.00),v40,z0,tPen\WObj:=wPaper;
    MoveL Offs(pOrigin,175.10,52.66,0.00),v40,z0,tPen\WObj:=wPaper;
    MoveL Offs(pOrigin,198.50,52.66,0.00),v40,z0,tPen\WObj:=wPaper;
    MoveL Offs(pOrigin,198.50,53.72,0.00),v40,z0,tPen\WObj:=wPaper;
    MoveL Offs(pOrigin,175.10,53.72,0.00),v40,z0,tPen\WObj:=wPaper;
    MoveL Offs(pOrigin,175.10,54.78,0.00),v40,z0,tPen\WObj:=wPaper;
    MoveL Offs(pOrigin,198.50,54.78,0.00),v40,z0,tPen\WObj:=wPaper;
    MoveL Offs(pOrigin,198.50,55.83,0.00),v40,z0,tPen\WObj:=wPaper;
    MoveL Offs(pOrigin,175.25,55.83,0.00),v40,z0,tPen\WObj:=wPaper;
    MoveL Offs(pOrigin,175.10,56.89,0.00),v40,z0,tPen\WObj:=wPaper;
    MoveL Offs(pOrigin,198.50,56.89,0.00),v40,z0,tPen\WObj:=wPaper;
    MoveL Offs(pOrigin,199.18,56.97,0.00),v40,z0,tPen\WObj:=wPaper;
    MoveL Offs(pOrigin,192.92,50.71,0.00),v40,fine,tPen\WObj:=wPaper;
    MoveL Offs(pOrigin,192.92,50.71,6.00),v60,z5,tPen\WObj:=wPaper;
    MoveL Offs(pOrigin,193.55,49.51,6.00),vTravel,z5,tPen\WObj:=wPaper;
    MoveL Offs(pOrigin,193.55,49.51,0.00),v60,z0,tPen\WObj:=wPaper;
    MoveL Offs(pOrigin,173.18,69.88,0.00),v40,z0,tPen\WObj:=wPaper;
    MoveL Offs(pOrigin,174.26,69.38,0.00),v40,z0,tPen\WObj:=wPaper;
    MoveL Offs(pOrigin,195.15,90.28,0.00),v40,z0,tPen\WObj:=wPaper;
    MoveL Offs(pOrigin,195.58,90.79,0.00),v40,z0,tPen\WObj:=wPaper;
    MoveL Offs(pOrigin,199.61,86.76,0.00),v40,z0,tPen\WObj:=wPaper;
    MoveL Offs(pOrigin,199.10,86.75,0.00),v40,z0,tPen\WObj:=wPaper;
    MoveL Offs(pOrigin,174.28,61.93,0.00),v40,z0,tPen\WObj:=wPaper;
    MoveL Offs(pOrigin,175.10,62.17,0.00),v40,z0,tPen\WObj:=wPaper;
    MoveL Offs(pOrigin,198.35,62.17,0.00),v40,z0,tPen\WObj:=wPaper;
    MoveL Offs(pOrigin,198.35,61.11,0.00),v40,z0,tPen\WObj:=wPaper;
    MoveL Offs(pOrigin,175.10,61.11,0.00),v40,z0,tPen\WObj:=wPaper;
    MoveL Offs(pOrigin,174.28,60.45,0.00),v40,z0,tPen\WObj:=wPaper;
    MoveL Offs(pOrigin,199.10,85.27,0.00),v40,z0,tPen\WObj:=wPaper;
    MoveL Offs(pOrigin,199.82,85.06,0.00),v40,z0,tPen\WObj:=wPaper;
    MoveL Offs(pOrigin,193.77,91.10,0.00),v40,z0,tPen\WObj:=wPaper;
    MoveL Offs(pOrigin,193.88,90.49,0.00),v40,z0,tPen\WObj:=wPaper;
    MoveL Offs(pOrigin,174.25,70.87,0.00),v40,z0,tPen\WObj:=wPaper;
    MoveL Offs(pOrigin,173.40,71.15,0.00),v40,z0,tPen\WObj:=wPaper;
    MoveL Offs(pOrigin,194.83,49.73,0.00),v40,z0,tPen\WObj:=wPaper;
    MoveL Offs(pOrigin,194.41,50.71,0.00),v40,z0,tPen\WObj:=wPaper;
    MoveL Offs(pOrigin,199.40,55.69,0.00),v40,z0,tPen\WObj:=wPaper;
    MoveL Offs(pOrigin,200.27,56.23,0.00),v40,z0,tPen\WObj:=wPaper;
    MoveL Offs(pOrigin,173.22,83.28,0.00),v40,z0,tPen\WObj:=wPaper;
    MoveL Offs(pOrigin,174.22,82.78,0.00),v40,z0,tPen\WObj:=wPaper;
    MoveL Offs(pOrigin,181.96,90.53,0.00),v40,z0,tPen\WObj:=wPaper;
    MoveL Offs(pOrigin,181.86,91.07,0.00),v40,z0,tPen\WObj:=wPaper;
    MoveL Offs(pOrigin,199.57,73.36,0.00),v40,z0,tPen\WObj:=wPaper;
    MoveL Offs(pOrigin,199.14,73.35,0.00),v40,z0,tPen\WObj:=wPaper;
    MoveL Offs(pOrigin,176.54,50.76,0.00),v40,z0,tPen\WObj:=wPaper;
    MoveL Offs(pOrigin,176.96,49.68,0.00),v40,z0,tPen\WObj:=wPaper;
    MoveL Offs(pOrigin,173.46,53.18,0.00),v40,z0,tPen\WObj:=wPaper;
    MoveL Offs(pOrigin,174.30,53.00,0.00),v40,z0,tPen\WObj:=wPaper;
    MoveL Offs(pOrigin,199.12,77.82,0.00),v40,z0,tPen\WObj:=wPaper;
    MoveL Offs(pOrigin,199.80,77.61,0.00),v40,z0,tPen\WObj:=wPaper;
    MoveL Offs(pOrigin,173.18,104.23,0.00),v40,fine,tPen\WObj:=wPaper;
    MoveL Offs(pOrigin,173.18,104.23,6.00),v60,z5,tPen\WObj:=wPaper;
    MoveL Offs(pOrigin,173.38,102.53,6.00),vTravel,z5,tPen\WObj:=wPaper;
    MoveL Offs(pOrigin,173.38,102.53,0.00),v60,z0,tPen\WObj:=wPaper;
    MoveL Offs(pOrigin,183.88,92.03,0.00),v40,z0,tPen\WObj:=wPaper;
    MoveL Offs(pOrigin,184.40,92.97,0.00),v40,z0,tPen\WObj:=wPaper;
  ENDPROC

  PROC DrawPart29()
    MoveL Offs(pOrigin,199.04,107.60,0.00),v40,z0,tPen\WObj:=wPaper;
    MoveL Offs(pOrigin,198.50,107.58,0.00),v40,z0,tPen\WObj:=wPaper;
    MoveL Offs(pOrigin,175.10,107.58,0.00),v40,z0,tPen\WObj:=wPaper;
    MoveL Offs(pOrigin,175.10,108.63,0.00),v40,z0,tPen\WObj:=wPaper;
    MoveL Offs(pOrigin,198.35,108.63,0.00),v40,z0,tPen\WObj:=wPaper;
    MoveL Offs(pOrigin,199.14,109.20,0.00),v40,z0,tPen\WObj:=wPaper;
    MoveL Offs(pOrigin,182.81,92.86,0.00),v40,z0,tPen\WObj:=wPaper;
    MoveL Offs(pOrigin,182.18,92.24,0.00),v40,z0,tPen\WObj:=wPaper;
    MoveL Offs(pOrigin,173.48,100.94,0.00),v40,z0,tPen\WObj:=wPaper;
    MoveL Offs(pOrigin,174.17,100.65,0.00),v40,z0,tPen\WObj:=wPaper;
    MoveL Offs(pOrigin,199.41,125.90,0.00),v40,z0,tPen\WObj:=wPaper;
    MoveL Offs(pOrigin,198.65,125.53,0.00),v40,z0,tPen\WObj:=wPaper;
    MoveL Offs(pOrigin,175.25,125.53,0.00),v40,z0,tPen\WObj:=wPaper;
    MoveL Offs(pOrigin,175.25,124.47,0.00),v40,z0,tPen\WObj:=wPaper;
    MoveL Offs(pOrigin,198.50,124.47,0.00),v40,z0,tPen\WObj:=wPaper;
    MoveL Offs(pOrigin,198.50,123.42,0.00),v40,z0,tPen\WObj:=wPaper;
    MoveL Offs(pOrigin,175.25,123.42,0.00),v40,z0,tPen\WObj:=wPaper;
    MoveL Offs(pOrigin,174.32,123.20,0.00),v40,z0,tPen\WObj:=wPaper;
    MoveL Offs(pOrigin,184.39,133.28,0.00),v40,z0,tPen\WObj:=wPaper;
    MoveL Offs(pOrigin,183.79,133.94,0.00),v40,z0,tPen\WObj:=wPaper;
    MoveL Offs(pOrigin,199.91,117.82,0.00),v40,fine,tPen\WObj:=wPaper;
    MoveL Offs(pOrigin,199.91,117.82,6.00),v60,z5,tPen\WObj:=wPaper;
    MoveL Offs(pOrigin,201.30,117.93,6.00),vTravel,z5,tPen\WObj:=wPaper;
    MoveL Offs(pOrigin,201.30,117.93,0.00),v60,z0,tPen\WObj:=wPaper;
    MoveL Offs(pOrigin,226.96,92.26,0.00),v40,z0,tPen\WObj:=wPaper;
    MoveL Offs(pOrigin,227.39,93.33,0.00),v40,z0,tPen\WObj:=wPaper;
    MoveL Offs(pOrigin,221.13,99.58,0.00),v40,z0,tPen\WObj:=wPaper;
    MoveL Offs(pOrigin,220.55,99.24,0.00),v40,z0,tPen\WObj:=wPaper;
    MoveL Offs(pOrigin,214.18,92.88,0.00),v40,z0,tPen\WObj:=wPaper;
    MoveL Offs(pOrigin,213.67,92.12,0.00),v40,z0,tPen\WObj:=wPaper;
    MoveL Offs(pOrigin,201.47,104.31,0.00),v40,z0,tPen\WObj:=wPaper;
    MoveL Offs(pOrigin,202.03,104.62,0.00),v40,z0,tPen\WObj:=wPaper;
    MoveL Offs(pOrigin,222.39,124.98,0.00),v40,z0,tPen\WObj:=wPaper;
    MoveL Offs(pOrigin,221.90,125.62,0.00),v40,z0,tPen\WObj:=wPaper;
    MoveL Offs(pOrigin,221.30,126.38,0.00),v40,z0,tPen\WObj:=wPaper;
    MoveL Offs(pOrigin,221.90,125.62,0.00),v40,z0,tPen\WObj:=wPaper;
    MoveL Offs(pOrigin,221.75,125.83,0.00),v40,z0,tPen\WObj:=wPaper;
    MoveL Offs(pOrigin,202.02,106.11,0.00),v40,z0,tPen\WObj:=wPaper;
    MoveL Offs(pOrigin,201.47,105.80,0.00),v40,z0,tPen\WObj:=wPaper;
    MoveL Offs(pOrigin,215.16,92.12,0.00),v40,z0,tPen\WObj:=wPaper;
    MoveL Offs(pOrigin,215.67,92.88,0.00),v40,z0,tPen\WObj:=wPaper;
    MoveL Offs(pOrigin,221.51,98.71,0.00),v40,z0,tPen\WObj:=wPaper;
    MoveL Offs(pOrigin,221.00,98.07,0.00),v40,z0,tPen\WObj:=wPaper;
    MoveL Offs(pOrigin,202.70,98.07,0.00),v40,z0,tPen\WObj:=wPaper;
    MoveL Offs(pOrigin,202.04,98.66,0.00),v40,z0,tPen\WObj:=wPaper;
    MoveL Offs(pOrigin,224.21,120.83,0.00),v40,z0,tPen\WObj:=wPaper;
    MoveL Offs(pOrigin,223.55,120.25,0.00),v40,z0,tPen\WObj:=wPaper;
    MoveL Offs(pOrigin,203.00,120.25,0.00),v40,z0,tPen\WObj:=wPaper;
    MoveL Offs(pOrigin,202.85,121.30,0.00),v40,z0,tPen\WObj:=wPaper;
    MoveL Offs(pOrigin,223.25,121.30,0.00),v40,z0,tPen\WObj:=wPaper;
    MoveL Offs(pOrigin,222.80,122.36,0.00),v40,z0,tPen\WObj:=wPaper;
    MoveL Offs(pOrigin,202.85,122.36,0.00),v40,z0,tPen\WObj:=wPaper;
    MoveL Offs(pOrigin,202.08,122.59,0.00),v40,z0,tPen\WObj:=wPaper;
    MoveL Offs(pOrigin,212.26,132.77,0.00),v40,z0,tPen\WObj:=wPaper;
    MoveL Offs(pOrigin,212.61,133.49,0.00),v40,z0,tPen\WObj:=wPaper;
    MoveL Offs(pOrigin,225.24,120.87,0.00),v40,fine,tPen\WObj:=wPaper;
    MoveL Offs(pOrigin,225.24,120.87,6.00),v60,z5,tPen\WObj:=wPaper;
    MoveL Offs(pOrigin,225.55,119.06,6.00),vTravel,z5,tPen\WObj:=wPaper;
    MoveL Offs(pOrigin,225.55,119.06,0.00),v60,z0,tPen\WObj:=wPaper;
    MoveL Offs(pOrigin,210.91,133.70,0.00),v40,z0,tPen\WObj:=wPaper;
    MoveL Offs(pOrigin,210.88,132.88,0.00),v40,z0,tPen\WObj:=wPaper;
    MoveL Offs(pOrigin,202.08,124.08,0.00),v40,z0,tPen\WObj:=wPaper;
    MoveL Offs(pOrigin,202.85,124.47,0.00),v40,z0,tPen\WObj:=wPaper;
    MoveL Offs(pOrigin,221.60,124.47,0.00),v40,fine,tPen\WObj:=wPaper;
    MoveL Offs(pOrigin,221.60,124.47,6.00),v60,z5,tPen\WObj:=wPaper;
    MoveL Offs(pOrigin,221.00,125.53,6.00),vTravel,z5,tPen\WObj:=wPaper;
    MoveL Offs(pOrigin,221.00,125.53,0.00),v60,z0,tPen\WObj:=wPaper;
    MoveL Offs(pOrigin,202.85,125.53,0.00),v40,z0,tPen\WObj:=wPaper;
    MoveL Offs(pOrigin,201.86,125.36,0.00),v40,z0,tPen\WObj:=wPaper;
    MoveL Offs(pOrigin,209.71,133.21,0.00),v40,z0,tPen\WObj:=wPaper;
    MoveL Offs(pOrigin,209.11,134.01,0.00),v40,z0,tPen\WObj:=wPaper;
    MoveL Offs(pOrigin,225.97,117.15,0.00),v40,fine,tPen\WObj:=wPaper;
    MoveL Offs(pOrigin,225.97,117.15,6.00),v60,z5,tPen\WObj:=wPaper;
    MoveL Offs(pOrigin,224.15,116.02,6.00),vTravel,z5,tPen\WObj:=wPaper;
    MoveL Offs(pOrigin,224.15,116.02,0.00),v60,z0,tPen\WObj:=wPaper;
    MoveL Offs(pOrigin,203.00,116.02,0.00),v40,z0,tPen\WObj:=wPaper;
    MoveL Offs(pOrigin,203.15,114.97,0.00),v40,z0,tPen\WObj:=wPaper;
    MoveL Offs(pOrigin,224.15,114.97,0.00),v40,fine,tPen\WObj:=wPaper;
    MoveL Offs(pOrigin,224.15,114.97,6.00),v60,z5,tPen\WObj:=wPaper;
    MoveL Offs(pOrigin,225.96,114.17,6.00),vTravel,z5,tPen\WObj:=wPaper;
    MoveL Offs(pOrigin,225.96,114.17,0.00),v60,z0,tPen\WObj:=wPaper;
    MoveL Offs(pOrigin,205.92,134.22,0.00),v40,z0,tPen\WObj:=wPaper;
    MoveL Offs(pOrigin,205.35,133.33,0.00),v40,z0,tPen\WObj:=wPaper;
    MoveL Offs(pOrigin,201.85,129.83,0.00),v40,z0,tPen\WObj:=wPaper;
    MoveL Offs(pOrigin,202.70,129.75,0.00),v40,z0,tPen\WObj:=wPaper;
    MoveL Offs(pOrigin,216.50,129.75,0.00),v40,fine,tPen\WObj:=wPaper;
    MoveL Offs(pOrigin,216.50,129.75,6.00),v60,z5,tPen\WObj:=wPaper;
    MoveL Offs(pOrigin,217.85,128.70,6.00),vTravel,z5,tPen\WObj:=wPaper;
    MoveL Offs(pOrigin,217.85,128.70,0.00),v60,z0,tPen\WObj:=wPaper;
    MoveL Offs(pOrigin,202.85,128.70,0.00),v40,z0,tPen\WObj:=wPaper;
    MoveL Offs(pOrigin,202.85,127.64,0.00),v40,z0,tPen\WObj:=wPaper;
    MoveL Offs(pOrigin,219.05,127.64,0.00),v40,fine,tPen\WObj:=wPaper;
    MoveL Offs(pOrigin,219.05,127.64,6.00),v60,z5,tPen\WObj:=wPaper;
    MoveL Offs(pOrigin,220.10,126.58,6.00),vTravel,z5,tPen\WObj:=wPaper;
    MoveL Offs(pOrigin,220.10,126.58,0.00),v60,z0,tPen\WObj:=wPaper;
    MoveL Offs(pOrigin,202.85,126.58,0.00),v40,z0,tPen\WObj:=wPaper;
    MoveL Offs(pOrigin,201.86,126.85,0.00),v40,z0,tPen\WObj:=wPaper;
    MoveL Offs(pOrigin,208.33,133.32,0.00),v40,fine,tPen\WObj:=wPaper;
    MoveL Offs(pOrigin,208.33,133.32,6.00),v60,z5,tPen\WObj:=wPaper;
    MoveL Offs(pOrigin,204.64,134.00,6.00),vTravel,z5,tPen\WObj:=wPaper;
    MoveL Offs(pOrigin,204.64,134.00,0.00),v60,z0,tPen\WObj:=wPaper;
    MoveL Offs(pOrigin,225.64,113.00,0.00),v40,fine,tPen\WObj:=wPaper;
    MoveL Offs(pOrigin,225.64,113.00,6.00),v60,z5,tPen\WObj:=wPaper;
    MoveL Offs(pOrigin,225.21,110.45,6.00),vTravel,z5,tPen\WObj:=wPaper;
    MoveL Offs(pOrigin,225.21,110.45,0.00),v60,z0,tPen\WObj:=wPaper;
    MoveL Offs(pOrigin,201.98,133.67,0.00),v40,z0,tPen\WObj:=wPaper;
    MoveL Offs(pOrigin,200.91,133.25,0.00),v40,z0,tPen\WObj:=wPaper;
    MoveL Offs(pOrigin,224.88,109.27,0.00),v40,z0,tPen\WObj:=wPaper;
    MoveL Offs(pOrigin,224.46,108.21,0.00),v40,z0,tPen\WObj:=wPaper;
    MoveL Offs(pOrigin,198.68,133.98,0.00),v40,fine,tPen\WObj:=wPaper;
    MoveL Offs(pOrigin,198.68,133.98,6.00),v60,z5,tPen\WObj:=wPaper;
    MoveL Offs(pOrigin,198.65,131.86,6.00),vTravel,z5,tPen\WObj:=wPaper;
    MoveL Offs(pOrigin,198.65,131.86,0.00),v60,z0,tPen\WObj:=wPaper;
    MoveL Offs(pOrigin,175.25,131.86,0.00),v40,z0,tPen\WObj:=wPaper;
    MoveL Offs(pOrigin,174.29,132.14,0.00),v40,z0,tPen\WObj:=wPaper;
    MoveL Offs(pOrigin,175.35,133.20,0.00),v40,z0,tPen\WObj:=wPaper;
    MoveL Offs(pOrigin,174.96,133.81,0.00),v40,z0,tPen\WObj:=wPaper;
    MoveL Offs(pOrigin,199.57,109.20,0.00),v40,z0,tPen\WObj:=wPaper;
    MoveL Offs(pOrigin,198.50,109.69,0.00),v40,z0,tPen\WObj:=wPaper;
    MoveL Offs(pOrigin,175.10,109.69,0.00),v40,z0,tPen\WObj:=wPaper;
  ENDPROC

  PROC DrawPart30()
    MoveL Offs(pOrigin,175.10,110.74,0.00),v40,z0,tPen\WObj:=wPaper;
    MoveL Offs(pOrigin,198.35,110.74,0.00),v40,z0,tPen\WObj:=wPaper;
    MoveL Offs(pOrigin,198.35,111.80,0.00),v40,z0,tPen\WObj:=wPaper;
    MoveL Offs(pOrigin,175.10,111.80,0.00),v40,z0,tPen\WObj:=wPaper;
    MoveL Offs(pOrigin,175.10,112.86,0.00),v40,z0,tPen\WObj:=wPaper;
    MoveL Offs(pOrigin,198.35,112.86,0.00),v40,z0,tPen\WObj:=wPaper;
    MoveL Offs(pOrigin,199.24,112.28,0.00),v40,z0,tPen\WObj:=wPaper;
    MoveL Offs(pOrigin,179.83,92.87,0.00),v40,fine,tPen\WObj:=wPaper;
    MoveL Offs(pOrigin,179.83,92.87,6.00),v60,z5,tPen\WObj:=wPaper;
    MoveL Offs(pOrigin,178.34,92.88,6.00),vTravel,z5,tPen\WObj:=wPaper;
    MoveL Offs(pOrigin,178.34,92.88,0.00),v60,z0,tPen\WObj:=wPaper;
    MoveL Offs(pOrigin,199.13,113.67,0.00),v40,z0,tPen\WObj:=wPaper;
    MoveL Offs(pOrigin,199.79,113.46,0.00),v40,z0,tPen\WObj:=wPaper;
    MoveL Offs(pOrigin,179.11,134.14,0.00),v40,z0,tPen\WObj:=wPaper;
    MoveL Offs(pOrigin,178.44,133.30,0.00),v40,z0,tPen\WObj:=wPaper;
    MoveL Offs(pOrigin,174.30,129.16,0.00),v40,z0,tPen\WObj:=wPaper;
    MoveL Offs(pOrigin,173.46,129.34,0.00),v40,z0,tPen\WObj:=wPaper;
    MoveL Offs(pOrigin,199.87,102.93,0.00),v40,fine,tPen\WObj:=wPaper;
    MoveL Offs(pOrigin,199.87,102.93,6.00),v60,z5,tPen\WObj:=wPaper;
    MoveL Offs(pOrigin,199.65,101.65,6.00),vTravel,z5,tPen\WObj:=wPaper;
    MoveL Offs(pOrigin,199.65,101.65,0.00),v60,z0,tPen\WObj:=wPaper;
    MoveL Offs(pOrigin,173.46,127.85,0.00),v40,z0,tPen\WObj:=wPaper;
    MoveL Offs(pOrigin,174.30,127.67,0.00),v40,z0,tPen\WObj:=wPaper;
    MoveL Offs(pOrigin,179.93,133.29,0.00),v40,z0,tPen\WObj:=wPaper;
    MoveL Offs(pOrigin,180.60,134.14,0.00),v40,z0,tPen\WObj:=wPaper;
    MoveL Offs(pOrigin,199.59,115.16,0.00),v40,z0,tPen\WObj:=wPaper;
    MoveL Offs(pOrigin,199.12,115.15,0.00),v40,z0,tPen\WObj:=wPaper;
    MoveL Offs(pOrigin,176.85,92.88,0.00),v40,z0,tPen\WObj:=wPaper;
    MoveL Offs(pOrigin,176.33,92.12,0.00),v40,z0,tPen\WObj:=wPaper;
    MoveL Offs(pOrigin,173.57,94.87,0.00),v40,z0,tPen\WObj:=wPaper;
    MoveL Offs(pOrigin,174.18,94.70,0.00),v40,z0,tPen\WObj:=wPaper;
    MoveL Offs(pOrigin,199.22,119.73,0.00),v40,z0,tPen\WObj:=wPaper;
    MoveL Offs(pOrigin,199.92,119.31,0.00),v40,z0,tPen\WObj:=wPaper;
    MoveL Offs(pOrigin,185.07,134.16,0.00),v40,fine,tPen\WObj:=wPaper;
    MoveL Offs(pOrigin,185.07,134.16,6.00),v60,z5,tPen\WObj:=wPaper;
    MoveL Offs(pOrigin,182.80,133.18,6.00),vTravel,z5,tPen\WObj:=wPaper;
    MoveL Offs(pOrigin,182.80,133.18,0.00),v60,z0,tPen\WObj:=wPaper;
    MoveL Offs(pOrigin,174.31,124.69,0.00),v40,z0,tPen\WObj:=wPaper;
    MoveL Offs(pOrigin,173.23,125.08,0.00),v40,z0,tPen\WObj:=wPaper;
    MoveL Offs(pOrigin,199.96,98.35,0.00),v40,z0,tPen\WObj:=wPaper;
    MoveL Offs(pOrigin,199.28,98.88,0.00),v40,z0,tPen\WObj:=wPaper;
    MoveL Offs(pOrigin,193.55,93.15,0.00),v40,z0,tPen\WObj:=wPaper;
    MoveL Offs(pOrigin,194.10,92.27,0.00),v40,z0,tPen\WObj:=wPaper;
    MoveL Offs(pOrigin,173.41,112.96,0.00),v40,z0,tPen\WObj:=wPaper;
    MoveL Offs(pOrigin,174.24,112.67,0.00),v40,z0,tPen\WObj:=wPaper;
    MoveL Offs(pOrigin,194.92,133.36,0.00),v40,fine,tPen\WObj:=wPaper;
    MoveL Offs(pOrigin,194.92,133.36,6.00),v60,z5,tPen\WObj:=wPaper;
    MoveL Offs(pOrigin,195.90,131.18,6.00),vTravel,z5,tPen\WObj:=wPaper;
    MoveL Offs(pOrigin,195.90,131.18,0.00),v60,z0,tPen\WObj:=wPaper;
    MoveL Offs(pOrigin,195.90,125.18,0.00),v40,z0,tPen\WObj:=wPaper;
    MoveL Offs(pOrigin,194.84,125.18,0.00),v40,z0,tPen\WObj:=wPaper;
    MoveL Offs(pOrigin,194.84,128.77,0.00),v40,fine,tPen\WObj:=wPaper;
    MoveL Offs(pOrigin,194.84,128.77,6.00),v60,z5,tPen\WObj:=wPaper;
    MoveL Offs(pOrigin,193.78,127.28,6.00),vTravel,z5,tPen\WObj:=wPaper;
    MoveL Offs(pOrigin,193.78,127.28,0.00),v60,z0,tPen\WObj:=wPaper;
    MoveL Offs(pOrigin,193.78,125.32,0.00),v40,z0,tPen\WObj:=wPaper;
    MoveL Offs(pOrigin,192.73,125.48,0.00),v40,z0,tPen\WObj:=wPaper;
    MoveL Offs(pOrigin,192.73,126.82,0.00),v40,fine,tPen\WObj:=wPaper;
    MoveL Offs(pOrigin,192.73,126.82,6.00),v60,z5,tPen\WObj:=wPaper;
    MoveL Offs(pOrigin,196.95,125.02,6.00),vTravel,z5,tPen\WObj:=wPaper;
    MoveL Offs(pOrigin,196.95,125.02,0.00),v60,z0,tPen\WObj:=wPaper;
    MoveL Offs(pOrigin,196.95,131.32,0.00),v40,fine,tPen\WObj:=wPaper;
    MoveL Offs(pOrigin,196.95,131.32,6.00),v60,z5,tPen\WObj:=wPaper;
    MoveL Offs(pOrigin,198.65,129.75,6.00),vTravel,z5,tPen\WObj:=wPaper;
    MoveL Offs(pOrigin,198.65,129.75,0.00),v60,z0,tPen\WObj:=wPaper;
    MoveL Offs(pOrigin,175.10,129.75,0.00),v40,z0,tPen\WObj:=wPaper;
    MoveL Offs(pOrigin,175.10,128.70,0.00),v40,z0,tPen\WObj:=wPaper;
    MoveL Offs(pOrigin,198.65,128.70,0.00),v40,z0,tPen\WObj:=wPaper;
    MoveL Offs(pOrigin,198.65,127.64,0.00),v40,z0,tPen\WObj:=wPaper;
    MoveL Offs(pOrigin,175.25,127.64,0.00),v40,z0,tPen\WObj:=wPaper;
    MoveL Offs(pOrigin,175.25,126.58,0.00),v40,z0,tPen\WObj:=wPaper;
    MoveL Offs(pOrigin,198.65,126.58,0.00),v40,fine,tPen\WObj:=wPaper;
    MoveL Offs(pOrigin,198.65,126.58,6.00),v60,z5,tPen\WObj:=wPaper;
    MoveL Offs(pOrigin,200.25,124.95,6.00),vTravel,z5,tPen\WObj:=wPaper;
    MoveL Offs(pOrigin,200.25,124.95,0.00),v60,z0,tPen\WObj:=wPaper;
    MoveL Offs(pOrigin,191.02,134.17,0.00),v40,fine,tPen\WObj:=wPaper;
    MoveL Offs(pOrigin,191.02,134.17,6.00),v60,z5,tPen\WObj:=wPaper;
    MoveL Offs(pOrigin,191.94,133.36,6.00),vTravel,z5,tPen\WObj:=wPaper;
    MoveL Offs(pOrigin,191.94,133.36,0.00),v60,z0,tPen\WObj:=wPaper;
    MoveL Offs(pOrigin,174.23,115.65,0.00),v40,z0,tPen\WObj:=wPaper;
    MoveL Offs(pOrigin,173.53,115.83,0.00),v40,z0,tPen\WObj:=wPaper;
    MoveL Offs(pOrigin,196.97,92.39,0.00),v40,z0,tPen\WObj:=wPaper;
    MoveL Offs(pOrigin,196.53,93.14,0.00),v40,z0,tPen\WObj:=wPaper;
    MoveL Offs(pOrigin,199.18,95.80,0.00),v40,z0,tPen\WObj:=wPaper;
    MoveL Offs(pOrigin,198.50,95.96,0.00),v40,z0,tPen\WObj:=wPaper;
    MoveL Offs(pOrigin,174.95,95.96,0.00),v40,z0,tPen\WObj:=wPaper;
    MoveL Offs(pOrigin,174.95,97.02,0.00),v40,z0,tPen\WObj:=wPaper;
    MoveL Offs(pOrigin,198.65,97.02,0.00),v40,fine,tPen\WObj:=wPaper;
    MoveL Offs(pOrigin,198.65,97.02,6.00),v60,z5,tPen\WObj:=wPaper;
    MoveL Offs(pOrigin,199.96,96.86,6.00),vTravel,z5,tPen\WObj:=wPaper;
    MoveL Offs(pOrigin,199.96,96.86,0.00),v60,z0,tPen\WObj:=wPaper;
    MoveL Offs(pOrigin,173.44,123.38,0.00),v40,fine,tPen\WObj:=wPaper;
    MoveL Offs(pOrigin,173.44,123.38,6.00),v60,z5,tPen\WObj:=wPaper;
    MoveL Offs(pOrigin,175.10,122.36,6.00),vTravel,z5,tPen\WObj:=wPaper;
    MoveL Offs(pOrigin,175.10,122.36,0.00),v60,z0,tPen\WObj:=wPaper;
    MoveL Offs(pOrigin,198.35,122.36,0.00),v40,z0,tPen\WObj:=wPaper;
    MoveL Offs(pOrigin,198.35,121.30,0.00),v40,z0,tPen\WObj:=wPaper;
    MoveL Offs(pOrigin,175.10,121.30,0.00),v40,z0,tPen\WObj:=wPaper;
    MoveL Offs(pOrigin,175.10,120.25,0.00),v40,z0,tPen\WObj:=wPaper;
    MoveL Offs(pOrigin,198.50,120.25,0.00),v40,z0,tPen\WObj:=wPaper;
    MoveL Offs(pOrigin,198.50,119.19,0.00),v40,z0,tPen\WObj:=wPaper;
    MoveL Offs(pOrigin,175.10,119.19,0.00),v40,fine,tPen\WObj:=wPaper;
    MoveL Offs(pOrigin,175.10,119.19,6.00),v60,z5,tPen\WObj:=wPaper;
    MoveL Offs(pOrigin,174.22,120.12,6.00),vTravel,z5,tPen\WObj:=wPaper;
    MoveL Offs(pOrigin,174.22,120.12,0.00),v60,z0,tPen\WObj:=wPaper;
    MoveL Offs(pOrigin,187.48,133.38,0.00),v40,fine,tPen\WObj:=wPaper;
    MoveL Offs(pOrigin,187.48,133.38,6.00),v60,z5,tPen\WObj:=wPaper;
    MoveL Offs(pOrigin,187.45,131.02,6.00),vTravel,z5,tPen\WObj:=wPaper;
    MoveL Offs(pOrigin,187.45,131.02,0.00),v60,z0,tPen\WObj:=wPaper;
    MoveL Offs(pOrigin,187.45,127.88,0.00),v40,fine,tPen\WObj:=wPaper;
    MoveL Offs(pOrigin,187.45,127.88,6.00),v60,z5,tPen\WObj:=wPaper;
    MoveL Offs(pOrigin,186.39,126.98,6.00),vTravel,z5,tPen\WObj:=wPaper;
    MoveL Offs(pOrigin,186.39,126.98,0.00),v60,z0,tPen\WObj:=wPaper;
    MoveL Offs(pOrigin,186.39,131.02,0.00),v40,z0,tPen\WObj:=wPaper;
    MoveL Offs(pOrigin,185.34,130.88,0.00),v40,z0,tPen\WObj:=wPaper;
    MoveL Offs(pOrigin,185.34,126.98,0.00),v40,z0,tPen\WObj:=wPaper;
    MoveL Offs(pOrigin,184.28,127.42,0.00),v40,z0,tPen\WObj:=wPaper;
    MoveL Offs(pOrigin,184.28,130.88,0.00),v40,fine,tPen\WObj:=wPaper;
    MoveL Offs(pOrigin,184.28,130.88,6.00),v60,z5,tPen\WObj:=wPaper;
    MoveL Offs(pOrigin,183.22,130.12,6.00),vTravel,z5,tPen\WObj:=wPaper;
  ENDPROC

  PROC DrawPart31()
    MoveL Offs(pOrigin,183.22,130.12,0.00),v60,z0,tPen\WObj:=wPaper;
    MoveL Offs(pOrigin,183.22,128.02,0.00),v40,fine,tPen\WObj:=wPaper;
    MoveL Offs(pOrigin,183.22,128.02,6.00),v60,z5,tPen\WObj:=wPaper;
    MoveL Offs(pOrigin,188.50,129.22,6.00),vTravel,z5,tPen\WObj:=wPaper;
    MoveL Offs(pOrigin,188.50,129.22,0.00),v60,z0,tPen\WObj:=wPaper;
    MoveL Offs(pOrigin,188.50,131.02,0.00),v40,z0,tPen\WObj:=wPaper;
    MoveL Offs(pOrigin,189.56,131.18,0.00),v40,z0,tPen\WObj:=wPaper;
    MoveL Offs(pOrigin,189.56,130.27,0.00),v40,fine,tPen\WObj:=wPaper;
    MoveL Offs(pOrigin,189.56,130.27,6.00),v60,z5,tPen\WObj:=wPaper;
    MoveL Offs(pOrigin,192.51,134.18,6.00),vTravel,z5,tPen\WObj:=wPaper;
    MoveL Offs(pOrigin,192.51,134.18,0.00),v60,z0,tPen\WObj:=wPaper;
    MoveL Offs(pOrigin,222.11,104.59,0.00),v40,z0,tPen\WObj:=wPaper;
    MoveL Offs(pOrigin,222.75,105.44,0.00),v40,z0,tPen\WObj:=wPaper;
    MoveL Offs(pOrigin,201.00,127.18,0.00),v40,fine,tPen\WObj:=wPaper;
    MoveL Offs(pOrigin,201.00,127.18,6.00),v60,z5,tPen\WObj:=wPaper;
    MoveL Offs(pOrigin,201.10,124.10,6.00),vTravel,z5,tPen\WObj:=wPaper;
    MoveL Offs(pOrigin,201.10,124.10,0.00),v60,z0,tPen\WObj:=wPaper;
    MoveL Offs(pOrigin,221.46,103.73,0.00),v40,z0,tPen\WObj:=wPaper;
    MoveL Offs(pOrigin,220.85,104.32,0.00),v40,z0,tPen\WObj:=wPaper;
    MoveL Offs(pOrigin,221.45,104.93,0.00),v40,z0,tPen\WObj:=wPaper;
    MoveL Offs(pOrigin,220.85,104.32,0.00),v40,z0,tPen\WObj:=wPaper;
    MoveL Offs(pOrigin,219.95,104.41,0.00),v40,z0,tPen\WObj:=wPaper;
    MoveL Offs(pOrigin,202.85,104.41,0.00),v40,z0,tPen\WObj:=wPaper;
    MoveL Offs(pOrigin,202.85,105.46,0.00),v40,z0,tPen\WObj:=wPaper;
    MoveL Offs(pOrigin,220.85,105.46,0.00),v40,fine,tPen\WObj:=wPaper;
    MoveL Offs(pOrigin,220.85,105.46,6.00),v60,z5,tPen\WObj:=wPaper;
    MoveL Offs(pOrigin,221.60,106.52,6.00),vTravel,z5,tPen\WObj:=wPaper;
    MoveL Offs(pOrigin,221.60,106.52,0.00),v60,z0,tPen\WObj:=wPaper;
    MoveL Offs(pOrigin,203.00,106.52,0.00),v40,z0,tPen\WObj:=wPaper;
    MoveL Offs(pOrigin,203.00,107.58,0.00),v40,z0,tPen\WObj:=wPaper;
    MoveL Offs(pOrigin,222.35,107.58,0.00),v40,fine,tPen\WObj:=wPaper;
    MoveL Offs(pOrigin,222.35,107.58,6.00),v60,z5,tPen\WObj:=wPaper;
    MoveL Offs(pOrigin,222.20,105.97,6.00),vTravel,z5,tPen\WObj:=wPaper;
    MoveL Offs(pOrigin,222.20,105.97,0.00),v60,z0,tPen\WObj:=wPaper;
    MoveL Offs(pOrigin,222.50,106.43,0.00),v40,z0,tPen\WObj:=wPaper;
    MoveL Offs(pOrigin,222.20,105.97,0.00),v40,fine,tPen\WObj:=wPaper;
    MoveL Offs(pOrigin,222.20,105.97,6.00),v60,z5,tPen\WObj:=wPaper;
    MoveL Offs(pOrigin,220.61,103.09,6.00),vTravel,z5,tPen\WObj:=wPaper;
    MoveL Offs(pOrigin,220.61,103.09,0.00),v60,z0,tPen\WObj:=wPaper;
    MoveL Offs(pOrigin,201.41,122.29,0.00),v40,fine,tPen\WObj:=wPaper;
    MoveL Offs(pOrigin,201.41,122.29,6.00),v60,z5,tPen\WObj:=wPaper;
    MoveL Offs(pOrigin,202.08,121.10,6.00),vTravel,z5,tPen\WObj:=wPaper;
    MoveL Offs(pOrigin,202.08,121.10,0.00),v60,z0,tPen\WObj:=wPaper;
    MoveL Offs(pOrigin,213.33,132.35,0.00),v40,fine,tPen\WObj:=wPaper;
    MoveL Offs(pOrigin,213.33,132.35,6.00),v60,z5,tPen\WObj:=wPaper;
    MoveL Offs(pOrigin,211.85,131.86,6.00),vTravel,z5,tPen\WObj:=wPaper;
    MoveL Offs(pOrigin,211.85,131.86,0.00),v60,z0,tPen\WObj:=wPaper;
    MoveL Offs(pOrigin,202.85,131.86,0.00),v40,fine,tPen\WObj:=wPaper;
    MoveL Offs(pOrigin,202.85,131.86,6.00),v60,z5,tPen\WObj:=wPaper;
    MoveL Offs(pOrigin,208.57,129.07,6.00),vTravel,z5,tPen\WObj:=wPaper;
    MoveL Offs(pOrigin,208.57,129.07,0.00),v60,z0,tPen\WObj:=wPaper;
    MoveL Offs(pOrigin,208.57,127.58,0.00),v40,z0,tPen\WObj:=wPaper;
    MoveL Offs(pOrigin,209.62,128.02,0.00),v40,z0,tPen\WObj:=wPaper;
    MoveL Offs(pOrigin,209.62,129.68,0.00),v40,fine,tPen\WObj:=wPaper;
    MoveL Offs(pOrigin,209.62,129.68,6.00),v60,z5,tPen\WObj:=wPaper;
    MoveL Offs(pOrigin,202.85,123.42,6.00),vTravel,z5,tPen\WObj:=wPaper;
    MoveL Offs(pOrigin,202.85,123.42,0.00),v60,z0,tPen\WObj:=wPaper;
    MoveL Offs(pOrigin,222.20,123.42,0.00),v40,z0,tPen\WObj:=wPaper;
    MoveL Offs(pOrigin,222.92,124.02,0.00),v40,z0,tPen\WObj:=wPaper;
    MoveL Offs(pOrigin,202.03,103.13,0.00),v40,z0,tPen\WObj:=wPaper;
    MoveL Offs(pOrigin,201.47,102.83,0.00),v40,z0,tPen\WObj:=wPaper;
    MoveL Offs(pOrigin,211.97,92.32,0.00),v40,z0,tPen\WObj:=wPaper;
    MoveL Offs(pOrigin,211.42,93.10,0.00),v40,z0,tPen\WObj:=wPaper;
    MoveL Offs(pOrigin,218.74,100.42,0.00),v40,z0,tPen\WObj:=wPaper;
    MoveL Offs(pOrigin,217.85,100.18,0.00),v40,z0,tPen\WObj:=wPaper;
    MoveL Offs(pOrigin,202.85,100.18,0.00),v40,z0,tPen\WObj:=wPaper;
    MoveL Offs(pOrigin,202.85,101.24,0.00),v40,z0,tPen\WObj:=wPaper;
    MoveL Offs(pOrigin,217.40,101.24,0.00),v40,z0,tPen\WObj:=wPaper;
    MoveL Offs(pOrigin,218.41,101.59,0.00),v40,z0,tPen\WObj:=wPaper;
    MoveL Offs(pOrigin,209.93,93.11,0.00),v40,z0,tPen\WObj:=wPaper;
    MoveL Offs(pOrigin,210.37,92.43,0.00),v40,z0,tPen\WObj:=wPaper;
    MoveL Offs(pOrigin,201.57,101.23,0.00),v40,z0,tPen\WObj:=wPaper;
    MoveL Offs(pOrigin,202.03,101.64,0.00),v40,z0,tPen\WObj:=wPaper;
    MoveL Offs(pOrigin,223.46,123.06,0.00),v40,fine,tPen\WObj:=wPaper;
    MoveL Offs(pOrigin,223.46,123.06,6.00),v60,z5,tPen\WObj:=wPaper;
    MoveL Offs(pOrigin,222.17,126.92,6.00),vTravel,z5,tPen\WObj:=wPaper;
    MoveL Offs(pOrigin,222.17,126.92,0.00),v60,z0,tPen\WObj:=wPaper;
    MoveL Offs(pOrigin,221.43,127.67,0.00),v40,z0,tPen\WObj:=wPaper;
    MoveL Offs(pOrigin,221.21,126.79,0.00),v40,z0,tPen\WObj:=wPaper;
    MoveL Offs(pOrigin,202.12,107.70,0.00),v40,z0,tPen\WObj:=wPaper;
    MoveL Offs(pOrigin,201.48,107.29,0.00),v40,z0,tPen\WObj:=wPaper;
    MoveL Offs(pOrigin,216.54,92.23,0.00),v40,z0,tPen\WObj:=wPaper;
    MoveL Offs(pOrigin,216.11,91.17,0.00),v40,z0,tPen\WObj:=wPaper;
    MoveL Offs(pOrigin,233.19,74.09,0.00),v40,fine,tPen\WObj:=wPaper;
    MoveL Offs(pOrigin,233.19,74.09,6.00),v60,z5,tPen\WObj:=wPaper;
    MoveL Offs(pOrigin,232.97,72.81,6.00),vTravel,z5,tPen\WObj:=wPaper;
    MoveL Offs(pOrigin,232.97,72.81,0.00),v60,z0,tPen\WObj:=wPaper;
    MoveL Offs(pOrigin,214.52,91.27,0.00),v40,z0,tPen\WObj:=wPaper;
    MoveL Offs(pOrigin,214.72,90.43,0.00),v40,z0,tPen\WObj:=wPaper;
    MoveL Offs(pOrigin,202.21,77.92,0.00),v40,z0,tPen\WObj:=wPaper;
    MoveL Offs(pOrigin,201.39,77.51,0.00),v40,z0,tPen\WObj:=wPaper;
    MoveL Offs(pOrigin,223.03,55.87,0.00),v40,z0,tPen\WObj:=wPaper;
    MoveL Offs(pOrigin,222.39,55.02,0.00),v40,z0,tPen\WObj:=wPaper;
    MoveL Offs(pOrigin,201.39,76.02,0.00),v40,z0,tPen\WObj:=wPaper;
    MoveL Offs(pOrigin,202.21,76.43,0.00),v40,z0,tPen\WObj:=wPaper;
    MoveL Offs(pOrigin,216.21,90.43,0.00),v40,fine,tPen\WObj:=wPaper;
    MoveL Offs(pOrigin,216.21,90.43,6.00),v60,z5,tPen\WObj:=wPaper;
    MoveL Offs(pOrigin,217.70,90.42,6.00),vTravel,z5,tPen\WObj:=wPaper;
    MoveL Offs(pOrigin,217.70,90.42,0.00),v60,z0,tPen\WObj:=wPaper;
    MoveL Offs(pOrigin,202.22,74.94,0.00),v40,z0,tPen\WObj:=wPaper;
    MoveL Offs(pOrigin,201.49,74.43,0.00),v40,z0,tPen\WObj:=wPaper;
    MoveL Offs(pOrigin,221.54,54.38,0.00),v40,fine,tPen\WObj:=wPaper;
    MoveL Offs(pOrigin,221.54,54.38,6.00),v60,z5,tPen\WObj:=wPaper;
    MoveL Offs(pOrigin,219.62,53.31,6.00),vTravel,z5,tPen\WObj:=wPaper;
    MoveL Offs(pOrigin,219.62,53.31,0.00),v60,z0,tPen\WObj:=wPaper;
    MoveL Offs(pOrigin,201.48,71.45,0.00),v40,fine,tPen\WObj:=wPaper;
    MoveL Offs(pOrigin,201.48,71.45,6.00),v60,z5,tPen\WObj:=wPaper;
    MoveL Offs(pOrigin,203.30,71.67,6.00),vTravel,z5,tPen\WObj:=wPaper;
    MoveL Offs(pOrigin,203.30,71.67,0.00),v60,z0,tPen\WObj:=wPaper;
    MoveL Offs(pOrigin,230.90,71.67,0.00),v40,z0,tPen\WObj:=wPaper;
    MoveL Offs(pOrigin,231.05,72.73,0.00),v40,z0,tPen\WObj:=wPaper;
    MoveL Offs(pOrigin,203.15,72.73,0.00),v40,fine,tPen\WObj:=wPaper;
    MoveL Offs(pOrigin,203.15,72.73,6.00),v60,z5,tPen\WObj:=wPaper;
    MoveL Offs(pOrigin,203.15,74.84,6.00),vTravel,z5,tPen\WObj:=wPaper;
    MoveL Offs(pOrigin,203.15,74.84,0.00),v60,z0,tPen\WObj:=wPaper;
    MoveL Offs(pOrigin,231.35,74.84,0.00),v40,z0,tPen\WObj:=wPaper;
    MoveL Offs(pOrigin,232.21,75.07,0.00),v40,z0,tPen\WObj:=wPaper;
    MoveL Offs(pOrigin,207.82,50.67,0.00),v40,z0,tPen\WObj:=wPaper;
    MoveL Offs(pOrigin,208.33,49.66,0.00),v40,z0,tPen\WObj:=wPaper;
    MoveL Offs(pOrigin,201.23,56.77,0.00),v40,fine,tPen\WObj:=wPaper;
  ENDPROC

  PROC DrawPart32()
    MoveL Offs(pOrigin,201.23,56.77,6.00),v60,z5,tPen\WObj:=wPaper;
    MoveL Offs(pOrigin,199.85,58.15,6.00),vTravel,z5,tPen\WObj:=wPaper;
    MoveL Offs(pOrigin,199.85,58.15,0.00),v60,z0,tPen\WObj:=wPaper;
    MoveL Offs(pOrigin,173.44,84.56,0.00),v40,z0,tPen\WObj:=wPaper;
    MoveL Offs(pOrigin,174.32,84.38,0.00),v40,z0,tPen\WObj:=wPaper;
    MoveL Offs(pOrigin,180.47,90.53,0.00),v40,fine,tPen\WObj:=wPaper;
    MoveL Offs(pOrigin,180.47,90.53,6.00),v60,z5,tPen\WObj:=wPaper;
    MoveL Offs(pOrigin,178.98,90.53,6.00),vTravel,z5,tPen\WObj:=wPaper;
    MoveL Offs(pOrigin,178.98,90.53,0.00),v60,z0,tPen\WObj:=wPaper;
    MoveL Offs(pOrigin,174.32,85.87,0.00),v40,z0,tPen\WObj:=wPaper;
    MoveL Offs(pOrigin,173.55,85.94,0.00),v40,z0,tPen\WObj:=wPaper;
    MoveL Offs(pOrigin,199.85,59.64,0.00),v40,z0,tPen\WObj:=wPaper;
    MoveL Offs(pOrigin,199.17,59.95,0.00),v40,z0,tPen\WObj:=wPaper;
    MoveL Offs(pOrigin,190.05,50.83,0.00),v40,z0,tPen\WObj:=wPaper;
    MoveL Offs(pOrigin,190.36,49.72,0.00),v40,z0,tPen\WObj:=wPaper;
    MoveL Offs(pOrigin,173.49,66.58,0.00),v40,z0,tPen\WObj:=wPaper;
    MoveL Offs(pOrigin,174.27,66.40,0.00),v40,z0,tPen\WObj:=wPaper;
    MoveL Offs(pOrigin,198.13,90.27,0.00),v40,z0,tPen\WObj:=wPaper;
    MoveL Offs(pOrigin,198.56,90.80,0.00),v40,z0,tPen\WObj:=wPaper;
    MoveL Offs(pOrigin,199.83,89.52,0.00),v40,z0,tPen\WObj:=wPaper;
    MoveL Offs(pOrigin,199.09,89.73,0.00),v40,z0,tPen\WObj:=wPaper;
    MoveL Offs(pOrigin,174.27,64.91,0.00),v40,z0,tPen\WObj:=wPaper;
    MoveL Offs(pOrigin,173.49,65.09,0.00),v40,z0,tPen\WObj:=wPaper;
    MoveL Offs(pOrigin,188.87,49.71,0.00),v40,z0,tPen\WObj:=wPaper;
    MoveL Offs(pOrigin,188.56,50.83,0.00),v40,z0,tPen\WObj:=wPaper;
    MoveL Offs(pOrigin,199.17,61.44,0.00),v40,z0,tPen\WObj:=wPaper;
    MoveL Offs(pOrigin,199.86,61.12,0.00),v40,z0,tPen\WObj:=wPaper;
    MoveL Offs(pOrigin,173.55,87.43,0.00),v40,z0,tPen\WObj:=wPaper;
    MoveL Offs(pOrigin,174.31,87.36,0.00),v40,z0,tPen\WObj:=wPaper;
    MoveL Offs(pOrigin,177.49,90.54,0.00),v40,z0,tPen\WObj:=wPaper;
    MoveL Offs(pOrigin,177.18,91.27,0.00),v40,z0,tPen\WObj:=wPaper;
    MoveL Offs(pOrigin,199.88,68.57,0.00),v40,z0,tPen\WObj:=wPaper;
    MoveL Offs(pOrigin,199.04,68.78,0.00),v40,z0,tPen\WObj:=wPaper;
    MoveL Offs(pOrigin,181.01,50.75,0.00),v40,z0,tPen\WObj:=wPaper;
    MoveL Offs(pOrigin,181.32,49.80,0.00),v40,z0,tPen\WObj:=wPaper;
    MoveL Offs(pOrigin,173.47,57.65,0.00),v40,z0,tPen\WObj:=wPaper;
    MoveL Offs(pOrigin,174.29,57.47,0.00),v40,z0,tPen\WObj:=wPaper;
    MoveL Offs(pOrigin,199.11,82.29,0.00),v40,z0,tPen\WObj:=wPaper;
    MoveL Offs(pOrigin,199.81,82.08,0.00),v40,z0,tPen\WObj:=wPaper;
    MoveL Offs(pOrigin,191.01,90.88,0.00),v40,z0,tPen\WObj:=wPaper;
    MoveL Offs(pOrigin,190.90,90.50,0.00),v40,z0,tPen\WObj:=wPaper;
    MoveL Offs(pOrigin,174.24,73.85,0.00),v40,z0,tPen\WObj:=wPaper;
    MoveL Offs(pOrigin,173.51,74.03,0.00),v40,z0,tPen\WObj:=wPaper;
    MoveL Offs(pOrigin,197.80,49.74,0.00),v40,fine,tPen\WObj:=wPaper;
    MoveL Offs(pOrigin,197.80,49.74,6.00),v60,z5,tPen\WObj:=wPaper;
    MoveL Offs(pOrigin,199.08,49.95,6.00),vTravel,z5,tPen\WObj:=wPaper;
    MoveL Offs(pOrigin,199.08,49.95,0.00),v60,z0,tPen\WObj:=wPaper;
    MoveL Offs(pOrigin,173.20,75.83,0.00),v40,fine,tPen\WObj:=wPaper;
    MoveL Offs(pOrigin,173.20,75.83,6.00),v60,z5,tPen\WObj:=wPaper;
    MoveL Offs(pOrigin,174.24,76.83,6.00),vTravel,z5,tPen\WObj:=wPaper;
    MoveL Offs(pOrigin,174.24,76.83,0.00),v60,z0,tPen\WObj:=wPaper;
    MoveL Offs(pOrigin,187.92,90.51,0.00),v40,z0,tPen\WObj:=wPaper;
    MoveL Offs(pOrigin,187.82,91.09,0.00),v40,z0,tPen\WObj:=wPaper;
    MoveL Offs(pOrigin,199.59,79.31,0.00),v40,z0,tPen\WObj:=wPaper;
    MoveL Offs(pOrigin,199.12,79.31,0.00),v40,z0,tPen\WObj:=wPaper;
    MoveL Offs(pOrigin,174.30,54.49,0.00),v40,fine,tPen\WObj:=wPaper;
    MoveL Offs(pOrigin,174.30,54.49,6.00),v60,z5,tPen\WObj:=wPaper;
    MoveL Offs(pOrigin,173.14,54.99,6.00),vTravel,z5,tPen\WObj:=wPaper;
    MoveL Offs(pOrigin,173.14,54.99,0.00),v60,z0,tPen\WObj:=wPaper;
    MoveL Offs(pOrigin,178.76,49.36,0.00),v40,fine,tPen\WObj:=wPaper;
    MoveL Offs(pOrigin,178.76,49.36,6.00),v60,z5,tPen\WObj:=wPaper;
    MoveL Offs(pOrigin,177.93,50.65,6.00),vTravel,z5,tPen\WObj:=wPaper;
    MoveL Offs(pOrigin,177.93,50.65,0.00),v60,z0,tPen\WObj:=wPaper;
    MoveL Offs(pOrigin,199.14,71.86,0.00),v40,z0,tPen\WObj:=wPaper;
    MoveL Offs(pOrigin,199.57,71.87,0.00),v40,z0,tPen\WObj:=wPaper;
    MoveL Offs(pOrigin,173.16,98.28,0.00),v40,fine,tPen\WObj:=wPaper;
    MoveL Offs(pOrigin,173.16,98.28,6.00),v60,z5,tPen\WObj:=wPaper;
    MoveL Offs(pOrigin,174.95,99.13,6.00),vTravel,z5,tPen\WObj:=wPaper;
    MoveL Offs(pOrigin,174.95,99.13,0.00),v60,z0,tPen\WObj:=wPaper;
    MoveL Offs(pOrigin,198.65,99.13,0.00),v40,z0,tPen\WObj:=wPaper;
    MoveL Offs(pOrigin,198.65,100.18,0.00),v40,z0,tPen\WObj:=wPaper;
    MoveL Offs(pOrigin,174.95,100.18,0.00),v40,z0,tPen\WObj:=wPaper;
    MoveL Offs(pOrigin,174.95,101.24,0.00),v40,z0,tPen\WObj:=wPaper;
    MoveL Offs(pOrigin,198.50,101.24,0.00),v40,fine,tPen\WObj:=wPaper;
    MoveL Offs(pOrigin,198.50,101.24,6.00),v60,z5,tPen\WObj:=wPaper;
    MoveL Offs(pOrigin,196.95,101.78,6.00),vTravel,z5,tPen\WObj:=wPaper;
    MoveL Offs(pOrigin,196.95,101.78,0.00),v60,z0,tPen\WObj:=wPaper;
    MoveL Offs(pOrigin,196.95,98.18,0.00),v40,fine,tPen\WObj:=wPaper;
    MoveL Offs(pOrigin,196.95,98.18,6.00),v60,z5,tPen\WObj:=wPaper;
    MoveL Offs(pOrigin,195.90,97.28,6.00),vTravel,z5,tPen\WObj:=wPaper;
    MoveL Offs(pOrigin,195.90,97.28,0.00),v60,z0,tPen\WObj:=wPaper;
    MoveL Offs(pOrigin,195.90,103.72,0.00),v40,z0,tPen\WObj:=wPaper;
    MoveL Offs(pOrigin,194.84,104.02,0.00),v40,z0,tPen\WObj:=wPaper;
    MoveL Offs(pOrigin,194.84,96.82,0.00),v40,fine,tPen\WObj:=wPaper;
    MoveL Offs(pOrigin,194.84,96.82,6.00),v60,z5,tPen\WObj:=wPaper;
    MoveL Offs(pOrigin,193.78,95.92,6.00),vTravel,z5,tPen\WObj:=wPaper;
    MoveL Offs(pOrigin,193.78,95.92,0.00),v60,z0,tPen\WObj:=wPaper;
    MoveL Offs(pOrigin,193.78,104.18,0.00),v40,z0,tPen\WObj:=wPaper;
    MoveL Offs(pOrigin,192.73,104.48,0.00),v40,z0,tPen\WObj:=wPaper;
    MoveL Offs(pOrigin,192.73,95.18,0.00),v40,z0,tPen\WObj:=wPaper;
    MoveL Offs(pOrigin,191.67,94.88,0.00),v40,z0,tPen\WObj:=wPaper;
    MoveL Offs(pOrigin,191.67,104.62,0.00),v40,z0,tPen\WObj:=wPaper;
    MoveL Offs(pOrigin,190.62,104.92,0.00),v40,z0,tPen\WObj:=wPaper;
    MoveL Offs(pOrigin,190.62,94.88,0.00),v40,z0,tPen\WObj:=wPaper;
    MoveL Offs(pOrigin,189.56,94.88,0.00),v40,z0,tPen\WObj:=wPaper;
    MoveL Offs(pOrigin,189.56,104.48,0.00),v40,fine,tPen\WObj:=wPaper;
    MoveL Offs(pOrigin,189.56,104.48,6.00),v60,z5,tPen\WObj:=wPaper;
    MoveL Offs(pOrigin,188.50,103.58,6.00),vTravel,z5,tPen\WObj:=wPaper;
    MoveL Offs(pOrigin,188.50,103.58,0.00),v60,z0,tPen\WObj:=wPaper;
    MoveL Offs(pOrigin,188.50,94.88,0.00),v40,z0,tPen\WObj:=wPaper;
    MoveL Offs(pOrigin,187.45,94.88,0.00),v40,z0,tPen\WObj:=wPaper;
    MoveL Offs(pOrigin,187.45,102.38,0.00),v40,z0,tPen\WObj:=wPaper;
    MoveL Offs(pOrigin,186.39,102.22,0.00),v40,z0,tPen\WObj:=wPaper;
    MoveL Offs(pOrigin,186.39,95.78,0.00),v40,fine,tPen\WObj:=wPaper;
    MoveL Offs(pOrigin,186.39,95.78,6.00),v60,z5,tPen\WObj:=wPaper;
    MoveL Offs(pOrigin,185.34,97.72,6.00),vTravel,z5,tPen\WObj:=wPaper;
    MoveL Offs(pOrigin,185.34,97.72,0.00),v60,z0,tPen\WObj:=wPaper;
    MoveL Offs(pOrigin,185.34,101.92,0.00),v40,z0,tPen\WObj:=wPaper;
    MoveL Offs(pOrigin,184.28,102.22,0.00),v40,z0,tPen\WObj:=wPaper;
    MoveL Offs(pOrigin,184.28,98.32,0.00),v40,z0,tPen\WObj:=wPaper;
    MoveL Offs(pOrigin,183.22,97.88,0.00),v40,z0,tPen\WObj:=wPaper;
    MoveL Offs(pOrigin,183.22,102.98,0.00),v40,fine,tPen\WObj:=wPaper;
    MoveL Offs(pOrigin,183.22,102.98,6.00),v60,z5,tPen\WObj:=wPaper;
    MoveL Offs(pOrigin,183.22,104.62,6.00),vTravel,z5,tPen\WObj:=wPaper;
    MoveL Offs(pOrigin,183.22,104.62,0.00),v60,z0,tPen\WObj:=wPaper;
    MoveL Offs(pOrigin,183.22,107.32,0.00),v40,z0,tPen\WObj:=wPaper;
    MoveL Offs(pOrigin,182.17,107.78,0.00),v40,z0,tPen\WObj:=wPaper;
    MoveL Offs(pOrigin,182.17,96.68,0.00),v40,fine,tPen\WObj:=wPaper;
    MoveL Offs(pOrigin,182.17,96.68,6.00),v60,z5,tPen\WObj:=wPaper;
    MoveL Offs(pOrigin,181.11,95.92,6.00),vTravel,z5,tPen\WObj:=wPaper;
  ENDPROC

  PROC DrawPart33()
    MoveL Offs(pOrigin,181.11,95.92,0.00),v60,z0,tPen\WObj:=wPaper;
    MoveL Offs(pOrigin,181.11,108.22,0.00),v40,z0,tPen\WObj:=wPaper;
    MoveL Offs(pOrigin,180.06,108.38,0.00),v40,z0,tPen\WObj:=wPaper;
    MoveL Offs(pOrigin,180.06,95.02,0.00),v40,z0,tPen\WObj:=wPaper;
    MoveL Offs(pOrigin,179.00,94.72,0.00),v40,z0,tPen\WObj:=wPaper;
    MoveL Offs(pOrigin,179.00,106.88,0.00),v40,fine,tPen\WObj:=wPaper;
    MoveL Offs(pOrigin,179.00,106.88,6.00),v60,z5,tPen\WObj:=wPaper;
    MoveL Offs(pOrigin,177.94,105.82,6.00),vTravel,z5,tPen\WObj:=wPaper;
    MoveL Offs(pOrigin,177.94,105.82,0.00),v60,z0,tPen\WObj:=wPaper;
    MoveL Offs(pOrigin,177.94,94.72,0.00),v40,z0,tPen\WObj:=wPaper;
    MoveL Offs(pOrigin,176.89,94.72,0.00),v40,z0,tPen\WObj:=wPaper;
    MoveL Offs(pOrigin,176.89,105.08,0.00),v40,fine,tPen\WObj:=wPaper;
    MoveL Offs(pOrigin,176.89,105.08,6.00),v60,z5,tPen\WObj:=wPaper;
    MoveL Offs(pOrigin,175.10,106.52,6.00),vTravel,z5,tPen\WObj:=wPaper;
    MoveL Offs(pOrigin,175.10,106.52,0.00),v60,z0,tPen\WObj:=wPaper;
    MoveL Offs(pOrigin,198.50,106.52,0.00),v40,fine,tPen\WObj:=wPaper;
    MoveL Offs(pOrigin,198.50,106.52,6.00),v60,z5,tPen\WObj:=wPaper;
    MoveL Offs(pOrigin,199.88,105.91,6.00),vTravel,z5,tPen\WObj:=wPaper;
    MoveL Offs(pOrigin,199.88,105.91,0.00),v60,z0,tPen\WObj:=wPaper;
    MoveL Offs(pOrigin,173.26,132.53,0.00),v40,z0,tPen\WObj:=wPaper;
    MoveL Offs(pOrigin,173.79,133.49,0.00),v40,z0,tPen\WObj:=wPaper;
    MoveL Offs(pOrigin,199.67,107.61,0.00),v40,fine,tPen\WObj:=wPaper;
    MoveL Offs(pOrigin,199.67,107.61,6.00),v60,z5,tPen\WObj:=wPaper;
    MoveL Offs(pOrigin,201.38,110.38,6.00),vTravel,z5,tPen\WObj:=wPaper;
    MoveL Offs(pOrigin,201.38,110.38,0.00),v60,z0,tPen\WObj:=wPaper;
    MoveL Offs(pOrigin,233.20,78.56,0.00),v40,fine,tPen\WObj:=wPaper;
    MoveL Offs(pOrigin,233.20,78.56,6.00),v60,z5,tPen\WObj:=wPaper;
    MoveL Offs(pOrigin,232.41,79.75,6.00),vTravel,z5,tPen\WObj:=wPaper;
    MoveL Offs(pOrigin,232.41,79.75,0.00),v60,z0,tPen\WObj:=wPaper;
    MoveL Offs(pOrigin,203.45,50.79,0.00),v40,z0,tPen\WObj:=wPaper;
    MoveL Offs(pOrigin,203.55,49.97,0.00),v40,z0,tPen\WObj:=wPaper;
    MoveL Offs(pOrigin,201.32,52.19,0.00),v40,z0,tPen\WObj:=wPaper;
    MoveL Offs(pOrigin,202.07,52.39,0.00),v40,z0,tPen\WObj:=wPaper;
    MoveL Offs(pOrigin,231.98,82.30,0.00),v40,z0,tPen\WObj:=wPaper;
    MoveL Offs(pOrigin,231.05,82.23,0.00),v40,z0,tPen\WObj:=wPaper;
    MoveL Offs(pOrigin,203.15,82.23,0.00),v40,z0,tPen\WObj:=wPaper;
    MoveL Offs(pOrigin,203.15,81.18,0.00),v40,z0,tPen\WObj:=wPaper;
    MoveL Offs(pOrigin,231.20,81.18,0.00),v40,fine,tPen\WObj:=wPaper;
    MoveL Offs(pOrigin,231.20,81.18,6.00),v60,z5,tPen\WObj:=wPaper;
    MoveL Offs(pOrigin,230.90,83.29,6.00),vTravel,z5,tPen\WObj:=wPaper;
    MoveL Offs(pOrigin,230.90,83.29,0.00),v60,z0,tPen\WObj:=wPaper;
    MoveL Offs(pOrigin,203.00,83.29,0.00),v40,fine,tPen\WObj:=wPaper;
    MoveL Offs(pOrigin,203.00,83.29,6.00),v60,z5,tPen\WObj:=wPaper;
    MoveL Offs(pOrigin,202.41,81.11,6.00),vTravel,z5,tPen\WObj:=wPaper;
    MoveL Offs(pOrigin,202.41,81.11,0.00),v60,z0,tPen\WObj:=wPaper;
    MoveL Offs(pOrigin,211.75,90.44,0.00),v40,z0,tPen\WObj:=wPaper;
    MoveL Offs(pOrigin,211.86,90.94,0.00),v40,z0,tPen\WObj:=wPaper;
    MoveL Offs(pOrigin,232.43,70.37,0.00),v40,fine,tPen\WObj:=wPaper;
    MoveL Offs(pOrigin,232.43,70.37,6.00),v60,z5,tPen\WObj:=wPaper;
    MoveL Offs(pOrigin,230.60,70.62,6.00),vTravel,z5,tPen\WObj:=wPaper;
    MoveL Offs(pOrigin,230.60,70.62,0.00),v60,z0,tPen\WObj:=wPaper;
    MoveL Offs(pOrigin,203.30,70.62,0.00),v40,z0,tPen\WObj:=wPaper;
    MoveL Offs(pOrigin,203.15,69.56,0.00),v40,z0,tPen\WObj:=wPaper;
    MoveL Offs(pOrigin,230.30,69.56,0.00),v40,z0,tPen\WObj:=wPaper;
    MoveL Offs(pOrigin,230.00,68.50,0.00),v40,z0,tPen\WObj:=wPaper;
    MoveL Offs(pOrigin,203.15,68.50,0.00),v40,z0,tPen\WObj:=wPaper;
    MoveL Offs(pOrigin,203.15,67.45,0.00),v40,z0,tPen\WObj:=wPaper;
    MoveL Offs(pOrigin,229.70,67.45,0.00),v40,z0,tPen\WObj:=wPaper;
    MoveL Offs(pOrigin,229.25,66.39,0.00),v40,z0,tPen\WObj:=wPaper;
    MoveL Offs(pOrigin,203.15,66.39,0.00),v40,fine,tPen\WObj:=wPaper;
    MoveL Offs(pOrigin,203.15,66.39,6.00),v60,z5,tPen\WObj:=wPaper;
    MoveL Offs(pOrigin,199.66,65.80,6.00),vTravel,z5,tPen\WObj:=wPaper;
    MoveL Offs(pOrigin,199.66,65.80,0.00),v60,z0,tPen\WObj:=wPaper;
    MoveL Offs(pOrigin,174.52,90.94,0.00),v40,z0,tPen\WObj:=wPaper;
    MoveL Offs(pOrigin,173.67,90.30,0.00),v40,z0,tPen\WObj:=wPaper;
    MoveL Offs(pOrigin,199.87,64.10,0.00),v40,z0,tPen\WObj:=wPaper;
    MoveL Offs(pOrigin,199.06,64.31,0.00),v40,z0,tPen\WObj:=wPaper;
    MoveL Offs(pOrigin,185.48,50.73,0.00),v40,fine,tPen\WObj:=wPaper;
    MoveL Offs(pOrigin,185.48,50.73,6.00),v60,z5,tPen\WObj:=wPaper;
    MoveL Offs(pOrigin,183.99,50.74,6.00),vTravel,z5,tPen\WObj:=wPaper;
    MoveL Offs(pOrigin,183.99,50.74,0.00),v60,z0,tPen\WObj:=wPaper;
    MoveL Offs(pOrigin,199.05,65.80,0.00),v40,z0,tPen\WObj:=wPaper;
    MoveL Offs(pOrigin,198.20,65.34,0.00),v40,z0,tPen\WObj:=wPaper;
    MoveL Offs(pOrigin,175.10,65.34,0.00),v40,z0,tPen\WObj:=wPaper;
    MoveL Offs(pOrigin,175.25,64.28,0.00),v40,z0,tPen\WObj:=wPaper;
    MoveL Offs(pOrigin,198.35,64.28,0.00),v40,z0,tPen\WObj:=wPaper;
    MoveL Offs(pOrigin,198.35,63.22,0.00),v40,z0,tPen\WObj:=wPaper;
    MoveL Offs(pOrigin,175.10,63.22,0.00),v40,z0,tPen\WObj:=wPaper;
    MoveL Offs(pOrigin,174.27,63.42,0.00),v40,z0,tPen\WObj:=wPaper;
    MoveL Offs(pOrigin,199.09,88.24,0.00),v40,z0,tPen\WObj:=wPaper;
    MoveL Offs(pOrigin,199.62,88.25,0.00),v40,z0,tPen\WObj:=wPaper;
    MoveL Offs(pOrigin,197.07,90.79,0.00),v40,z0,tPen\WObj:=wPaper;
    MoveL Offs(pOrigin,196.64,90.27,0.00),v40,z0,tPen\WObj:=wPaper;
    MoveL Offs(pOrigin,174.26,67.89,0.00),v40,z0,tPen\WObj:=wPaper;
    MoveL Offs(pOrigin,173.39,68.18,0.00),v40,z0,tPen\WObj:=wPaper;
    MoveL Offs(pOrigin,192.06,49.51,0.00),v40,fine,tPen\WObj:=wPaper;
    MoveL Offs(pOrigin,192.06,49.51,6.00),v60,z5,tPen\WObj:=wPaper;
    MoveL Offs(pOrigin,191.44,50.72,6.00),vTravel,z5,tPen\WObj:=wPaper;
    MoveL Offs(pOrigin,191.44,50.72,0.00),v60,z0,tPen\WObj:=wPaper;
    MoveL Offs(pOrigin,199.18,58.46,0.00),v40,z0,tPen\WObj:=wPaper;
    MoveL Offs(pOrigin,198.35,57.94,0.00),v40,z0,tPen\WObj:=wPaper;
    MoveL Offs(pOrigin,175.10,57.94,0.00),v40,z0,tPen\WObj:=wPaper;
    MoveL Offs(pOrigin,175.10,59.00,0.00),v40,z0,tPen\WObj:=wPaper;
    MoveL Offs(pOrigin,198.35,59.00,0.00),v40,z0,tPen\WObj:=wPaper;
    MoveL Offs(pOrigin,198.35,60.06,0.00),v40,z0,tPen\WObj:=wPaper;
    MoveL Offs(pOrigin,175.10,60.06,0.00),v40,fine,tPen\WObj:=wPaper;
    MoveL Offs(pOrigin,175.10,60.06,6.00),v60,z5,tPen\WObj:=wPaper;
    MoveL Offs(pOrigin,174.29,58.96,6.00),vTravel,z5,tPen\WObj:=wPaper;
    MoveL Offs(pOrigin,174.29,58.96,0.00),v60,z0,tPen\WObj:=wPaper;
    MoveL Offs(pOrigin,199.11,83.78,0.00),v40,z0,tPen\WObj:=wPaper;
    MoveL Offs(pOrigin,199.81,83.57,0.00),v40,z0,tPen\WObj:=wPaper;
    MoveL Offs(pOrigin,192.28,91.10,0.00),v40,z0,tPen\WObj:=wPaper;
    MoveL Offs(pOrigin,192.39,90.50,0.00),v40,z0,tPen\WObj:=wPaper;
    MoveL Offs(pOrigin,174.25,72.36,0.00),v40,z0,tPen\WObj:=wPaper;
    MoveL Offs(pOrigin,173.51,72.54,0.00),v40,z0,tPen\WObj:=wPaper;
    MoveL Offs(pOrigin,196.10,49.95,0.00),v40,z0,tPen\WObj:=wPaper;
    MoveL Offs(pOrigin,196.01,50.81,0.00),v40,z0,tPen\WObj:=wPaper;
    MoveL Offs(pOrigin,199.40,54.20,0.00),v40,z0,tPen\WObj:=wPaper;
    MoveL Offs(pOrigin,200.26,54.74,0.00),v40,z0,tPen\WObj:=wPaper;
    MoveL Offs(pOrigin,173.43,81.58,0.00),v40,z0,tPen\WObj:=wPaper;
    MoveL Offs(pOrigin,174.22,81.29,0.00),v40,z0,tPen\WObj:=wPaper;
    MoveL Offs(pOrigin,183.45,90.52,0.00),v40,z0,tPen\WObj:=wPaper;
    MoveL Offs(pOrigin,183.35,91.07,0.00),v40,z0,tPen\WObj:=wPaper;
    MoveL Offs(pOrigin,199.58,74.85,0.00),v40,fine,tPen\WObj:=wPaper;
    MoveL Offs(pOrigin,199.58,74.85,6.00),v60,z5,tPen\WObj:=wPaper;
    MoveL Offs(pOrigin,198.35,73.78,6.00),vTravel,z5,tPen\WObj:=wPaper;
    MoveL Offs(pOrigin,198.35,73.78,0.00),v60,z0,tPen\WObj:=wPaper;
    MoveL Offs(pOrigin,175.25,73.78,0.00),v40,z0,tPen\WObj:=wPaper;
    MoveL Offs(pOrigin,175.25,72.73,0.00),v40,z0,tPen\WObj:=wPaper;
    MoveL Offs(pOrigin,198.35,72.73,0.00),v40,z0,tPen\WObj:=wPaper;
  ENDPROC

  PROC DrawPart34()
    MoveL Offs(pOrigin,198.35,71.67,0.00),v40,z0,tPen\WObj:=wPaper;
    MoveL Offs(pOrigin,175.25,71.67,0.00),v40,z0,tPen\WObj:=wPaper;
    MoveL Offs(pOrigin,175.25,70.62,0.00),v40,z0,tPen\WObj:=wPaper;
    MoveL Offs(pOrigin,198.35,70.62,0.00),v40,z0,tPen\WObj:=wPaper;
    MoveL Offs(pOrigin,198.35,69.56,0.00),v40,z0,tPen\WObj:=wPaper;
    MoveL Offs(pOrigin,175.25,69.56,0.00),v40,z0,tPen\WObj:=wPaper;
    MoveL Offs(pOrigin,175.25,68.50,0.00),v40,z0,tPen\WObj:=wPaper;
    MoveL Offs(pOrigin,198.20,68.50,0.00),v40,z0,tPen\WObj:=wPaper;
    MoveL Offs(pOrigin,198.20,67.45,0.00),v40,z0,tPen\WObj:=wPaper;
    MoveL Offs(pOrigin,175.25,67.45,0.00),v40,z0,tPen\WObj:=wPaper;
    MoveL Offs(pOrigin,175.25,66.39,0.00),v40,z0,tPen\WObj:=wPaper;
    MoveL Offs(pOrigin,198.20,66.39,0.00),v40,fine,tPen\WObj:=wPaper;
    MoveL Offs(pOrigin,198.20,66.39,6.00),v60,z5,tPen\WObj:=wPaper;
    MoveL Offs(pOrigin,199.05,67.29,6.00),vTravel,z5,tPen\WObj:=wPaper;
    MoveL Offs(pOrigin,199.05,67.29,0.00),v60,z0,tPen\WObj:=wPaper;
    MoveL Offs(pOrigin,182.50,50.74,0.00),v40,z0,tPen\WObj:=wPaper;
    MoveL Offs(pOrigin,182.81,49.80,0.00),v40,z0,tPen\WObj:=wPaper;
    MoveL Offs(pOrigin,173.47,59.13,0.00),v40,fine,tPen\WObj:=wPaper;
    MoveL Offs(pOrigin,173.47,59.13,6.00),v60,z5,tPen\WObj:=wPaper;
    MoveL Offs(pOrigin,173.37,60.73,6.00),vTravel,z5,tPen\WObj:=wPaper;
    MoveL Offs(pOrigin,173.37,60.73,0.00),v60,z0,tPen\WObj:=wPaper;
    MoveL Offs(pOrigin,184.61,49.49,0.00),v40,fine,tPen\WObj:=wPaper;
    MoveL Offs(pOrigin,184.61,49.49,6.00),v60,z5,tPen\WObj:=wPaper;
    MoveL Offs(pOrigin,186.31,49.28,6.00),vTravel,z5,tPen\WObj:=wPaper;
    MoveL Offs(pOrigin,186.31,49.28,0.00),v60,z0,tPen\WObj:=wPaper;
    MoveL Offs(pOrigin,173.16,62.43,0.00),v40,fine,tPen\WObj:=wPaper;
    MoveL Offs(pOrigin,173.16,62.43,6.00),v60,z5,tPen\WObj:=wPaper;
    MoveL Offs(pOrigin,173.38,63.71,6.00),vTravel,z5,tPen\WObj:=wPaper;
    MoveL Offs(pOrigin,173.38,63.71,0.00),v60,z0,tPen\WObj:=wPaper;
    MoveL Offs(pOrigin,187.49,49.60,0.00),v40,fine,tPen\WObj:=wPaper;
    MoveL Offs(pOrigin,187.49,49.60,6.00),v60,z5,tPen\WObj:=wPaper;
    MoveL Offs(pOrigin,186.97,50.73,6.00),vTravel,z5,tPen\WObj:=wPaper;
    MoveL Offs(pOrigin,186.97,50.73,0.00),v60,z0,tPen\WObj:=wPaper;
    MoveL Offs(pOrigin,199.17,62.93,0.00),v40,z0,tPen\WObj:=wPaper;
    MoveL Offs(pOrigin,199.97,62.51,0.00),v40,z0,tPen\WObj:=wPaper;
    MoveL Offs(pOrigin,173.45,89.02,0.00),v40,z0,tPen\WObj:=wPaper;
    MoveL Offs(pOrigin,174.31,88.85,0.00),v40,z0,tPen\WObj:=wPaper;
    MoveL Offs(pOrigin,175.90,90.44,0.00),v40,z0,tPen\WObj:=wPaper;
    MoveL Offs(pOrigin,175.80,91.16,0.00),v40,z0,tPen\WObj:=wPaper;
    MoveL Offs(pOrigin,199.66,67.29,0.00),v40,fine,tPen\WObj:=wPaper;
    MoveL Offs(pOrigin,199.66,67.29,6.00),v60,z5,tPen\WObj:=wPaper;
    MoveL Offs(pOrigin,201.45,59.53,6.00),vTravel,z5,tPen\WObj:=wPaper;
    MoveL Offs(pOrigin,201.45,59.53,0.00),v60,z0,tPen\WObj:=wPaper;
    MoveL Offs(pOrigin,210.78,50.20,0.00),v40,fine,tPen\WObj:=wPaper;
    MoveL Offs(pOrigin,210.78,50.20,6.00),v60,z5,tPen\WObj:=wPaper;
    MoveL Offs(pOrigin,213.95,52.66,6.00),vTravel,z5,tPen\WObj:=wPaper;
    MoveL Offs(pOrigin,213.95,52.66,0.00),v60,z0,tPen\WObj:=wPaper;
    MoveL Offs(pOrigin,202.85,52.66,0.00),v40,z0,tPen\WObj:=wPaper;
    MoveL Offs(pOrigin,202.85,53.72,0.00),v40,z0,tPen\WObj:=wPaper;
    MoveL Offs(pOrigin,216.65,53.72,0.00),v40,fine,tPen\WObj:=wPaper;
    MoveL Offs(pOrigin,216.65,53.72,6.00),v60,z5,tPen\WObj:=wPaper;
    MoveL Offs(pOrigin,218.75,53.92,6.00),vTravel,z5,tPen\WObj:=wPaper;
    MoveL Offs(pOrigin,218.75,53.92,0.00),v60,z0,tPen\WObj:=wPaper;
    MoveL Offs(pOrigin,219.20,54.22,0.00),v40,z0,tPen\WObj:=wPaper;
    MoveL Offs(pOrigin,218.75,53.92,0.00),v40,z0,tPen\WObj:=wPaper;
    MoveL Offs(pOrigin,218.60,54.78,0.00),v40,z0,tPen\WObj:=wPaper;
    MoveL Offs(pOrigin,202.85,54.78,0.00),v40,fine,tPen\WObj:=wPaper;
    MoveL Offs(pOrigin,202.85,54.78,6.00),v60,z5,tPen\WObj:=wPaper;
    MoveL Offs(pOrigin,199.94,52.08,6.00),vTravel,z5,tPen\WObj:=wPaper;
    MoveL Offs(pOrigin,199.94,52.08,0.00),v60,z0,tPen\WObj:=wPaper;
    MoveL Offs(pOrigin,173.42,78.60,0.00),v40,z0,tPen\WObj:=wPaper;
    MoveL Offs(pOrigin,174.23,78.32,0.00),v40,z0,tPen\WObj:=wPaper;
    MoveL Offs(pOrigin,186.54,90.62,0.00),v40,fine,tPen\WObj:=wPaper;
    MoveL Offs(pOrigin,186.54,90.62,6.00),v60,z5,tPen\WObj:=wPaper;
    MoveL Offs(pOrigin,188.30,89.62,6.00),vTravel,z5,tPen\WObj:=wPaper;
    MoveL Offs(pOrigin,188.30,89.62,0.00),v60,z0,tPen\WObj:=wPaper;
    MoveL Offs(pOrigin,175.85,89.62,0.00),v40,fine,tPen\WObj:=wPaper;
    MoveL Offs(pOrigin,175.85,89.62,6.00),v60,z5,tPen\WObj:=wPaper;
    MoveL Offs(pOrigin,175.25,88.57,6.00),vTravel,z5,tPen\WObj:=wPaper;
    MoveL Offs(pOrigin,175.25,88.57,0.00),v60,z0,tPen\WObj:=wPaper;
    MoveL Offs(pOrigin,198.35,88.57,0.00),v40,z0,tPen\WObj:=wPaper;
    MoveL Offs(pOrigin,198.35,87.51,0.00),v40,z0,tPen\WObj:=wPaper;
    MoveL Offs(pOrigin,175.25,87.51,0.00),v40,z0,tPen\WObj:=wPaper;
    MoveL Offs(pOrigin,175.25,86.46,0.00),v40,z0,tPen\WObj:=wPaper;
    MoveL Offs(pOrigin,198.35,86.46,0.00),v40,z0,tPen\WObj:=wPaper;
    MoveL Offs(pOrigin,198.35,85.40,0.00),v40,z0,tPen\WObj:=wPaper;
    MoveL Offs(pOrigin,175.25,85.40,0.00),v40,z0,tPen\WObj:=wPaper;
    MoveL Offs(pOrigin,175.25,84.34,0.00),v40,z0,tPen\WObj:=wPaper;
    MoveL Offs(pOrigin,198.20,84.34,0.00),v40,z0,tPen\WObj:=wPaper;
    MoveL Offs(pOrigin,198.35,83.29,0.00),v40,z0,tPen\WObj:=wPaper;
    MoveL Offs(pOrigin,175.25,83.29,0.00),v40,z0,tPen\WObj:=wPaper;
    MoveL Offs(pOrigin,175.25,82.23,0.00),v40,z0,tPen\WObj:=wPaper;
    MoveL Offs(pOrigin,198.35,82.23,0.00),v40,z0,tPen\WObj:=wPaper;
    MoveL Offs(pOrigin,198.20,81.18,0.00),v40,z0,tPen\WObj:=wPaper;
    MoveL Offs(pOrigin,175.25,81.18,0.00),v40,z0,tPen\WObj:=wPaper;
    MoveL Offs(pOrigin,175.25,80.12,0.00),v40,z0,tPen\WObj:=wPaper;
    MoveL Offs(pOrigin,198.20,80.12,0.00),v40,z0,tPen\WObj:=wPaper;
    MoveL Offs(pOrigin,198.20,79.06,0.00),v40,z0,tPen\WObj:=wPaper;
    MoveL Offs(pOrigin,175.25,79.06,0.00),v40,z0,tPen\WObj:=wPaper;
    MoveL Offs(pOrigin,175.25,78.01,0.00),v40,z0,tPen\WObj:=wPaper;
    MoveL Offs(pOrigin,198.20,78.01,0.00),v40,z0,tPen\WObj:=wPaper;
    MoveL Offs(pOrigin,198.20,76.95,0.00),v40,z0,tPen\WObj:=wPaper;
    MoveL Offs(pOrigin,175.25,76.95,0.00),v40,z0,tPen\WObj:=wPaper;
    MoveL Offs(pOrigin,175.25,75.90,0.00),v40,z0,tPen\WObj:=wPaper;
    MoveL Offs(pOrigin,198.20,75.90,0.00),v40,fine,tPen\WObj:=wPaper;
    MoveL Offs(pOrigin,198.20,75.90,6.00),v60,z5,tPen\WObj:=wPaper;
    MoveL Offs(pOrigin,201.50,78.89,6.00),vTravel,z5,tPen\WObj:=wPaper;
    MoveL Offs(pOrigin,201.50,78.89,0.00),v60,z0,tPen\WObj:=wPaper;
    MoveL Offs(pOrigin,223.88,56.51,0.00),v40,z0,tPen\WObj:=wPaper;
    MoveL Offs(pOrigin,223.40,57.12,0.00),v40,z0,tPen\WObj:=wPaper;
    MoveL Offs(pOrigin,225.65,59.33,0.00),v40,z0,tPen\WObj:=wPaper;
    MoveL Offs(pOrigin,223.40,57.12,0.00),v40,fine,tPen\WObj:=wPaper;
    MoveL Offs(pOrigin,223.40,57.12,6.00),v60,z5,tPen\WObj:=wPaper;
    MoveL Offs(pOrigin,224.74,57.15,6.00),vTravel,z5,tPen\WObj:=wPaper;
    MoveL Offs(pOrigin,224.74,57.15,0.00),v60,z0,tPen\WObj:=wPaper;
    MoveL Offs(pOrigin,201.51,80.38,0.00),v40,fine,tPen\WObj:=wPaper;
    MoveL Offs(pOrigin,201.51,80.38,6.00),v60,z5,tPen\WObj:=wPaper;
    MoveL Offs(pOrigin,203.15,76.95,6.00),vTravel,z5,tPen\WObj:=wPaper;
    MoveL Offs(pOrigin,203.15,76.95,0.00),v60,z0,tPen\WObj:=wPaper;
    MoveL Offs(pOrigin,231.50,76.95,0.00),v40,z0,tPen\WObj:=wPaper;
    MoveL Offs(pOrigin,231.35,75.90,0.00),v40,z0,tPen\WObj:=wPaper;
    MoveL Offs(pOrigin,203.15,75.90,0.00),v40,fine,tPen\WObj:=wPaper;
    MoveL Offs(pOrigin,203.15,75.90,6.00),v60,z5,tPen\WObj:=wPaper;
    MoveL Offs(pOrigin,203.00,86.46,6.00),vTravel,z5,tPen\WObj:=wPaper;
    MoveL Offs(pOrigin,203.00,86.46,0.00),v60,z0,tPen\WObj:=wPaper;
    MoveL Offs(pOrigin,230.15,86.46,0.00),v40,fine,tPen\WObj:=wPaper;
    MoveL Offs(pOrigin,230.15,86.46,6.00),v60,z5,tPen\WObj:=wPaper;
    MoveL Offs(pOrigin,232.37,85.36,6.00),vTravel,z5,tPen\WObj:=wPaper;
    MoveL Offs(pOrigin,232.37,85.36,0.00),v60,z0,tPen\WObj:=wPaper;
    MoveL Offs(pOrigin,201.50,116.23,0.00),v40,fine,tPen\WObj:=wPaper;
  ENDPROC

  PROC DrawPart35()
    MoveL Offs(pOrigin,201.50,116.23,6.00),v60,z5,tPen\WObj:=wPaper;
    MoveL Offs(pOrigin,199.80,116.44,6.00),vTravel,z5,tPen\WObj:=wPaper;
    MoveL Offs(pOrigin,199.80,116.44,0.00),v60,z0,tPen\WObj:=wPaper;
    MoveL Offs(pOrigin,182.30,133.94,0.00),v40,fine,tPen\WObj:=wPaper;
    MoveL Offs(pOrigin,182.30,133.94,6.00),v60,z5,tPen\WObj:=wPaper;
    MoveL Offs(pOrigin,181.31,133.18,6.00),vTravel,z5,tPen\WObj:=wPaper;
    MoveL Offs(pOrigin,181.31,133.18,0.00),v60,z0,tPen\WObj:=wPaper;
    MoveL Offs(pOrigin,174.31,126.18,0.00),v40,fine,tPen\WObj:=wPaper;
    MoveL Offs(pOrigin,174.31,126.18,6.00),v60,z5,tPen\WObj:=wPaper;
    MoveL Offs(pOrigin,173.25,131.04,6.00),vTravel,z5,tPen\WObj:=wPaper;
    MoveL Offs(pOrigin,173.25,131.04,0.00),v60,z0,tPen\WObj:=wPaper;
    MoveL Offs(pOrigin,199.98,104.31,0.00),v40,fine,tPen\WObj:=wPaper;
    MoveL Offs(pOrigin,199.98,104.31,6.00),v60,z5,tPen\WObj:=wPaper;
    MoveL Offs(pOrigin,202.85,103.35,6.00),vTravel,z5,tPen\WObj:=wPaper;
    MoveL Offs(pOrigin,202.85,103.35,0.00),v60,z0,tPen\WObj:=wPaper;
    MoveL Offs(pOrigin,218.90,103.35,0.00),v40,z0,tPen\WObj:=wPaper;
    MoveL Offs(pOrigin,219.80,103.12,0.00),v40,z0,tPen\WObj:=wPaper;
    MoveL Offs(pOrigin,220.55,103.88,0.00),v40,z0,tPen\WObj:=wPaper;
    MoveL Offs(pOrigin,219.80,103.12,0.00),v40,z0,tPen\WObj:=wPaper;
    MoveL Offs(pOrigin,219.76,102.45,0.00),v40,z0,tPen\WObj:=wPaper;
    MoveL Offs(pOrigin,201.41,120.80,0.00),v40,fine,tPen\WObj:=wPaper;
    MoveL Offs(pOrigin,201.41,120.80,6.00),v60,z5,tPen\WObj:=wPaper;
    MoveL Offs(pOrigin,201.30,119.42,6.00),vTravel,z5,tPen\WObj:=wPaper;
    MoveL Offs(pOrigin,201.30,119.42,0.00),v60,z0,tPen\WObj:=wPaper;
    MoveL Offs(pOrigin,219.22,101.49,0.00),v40,z0,tPen\WObj:=wPaper;
    MoveL Offs(pOrigin,218.60,102.07,0.00),v40,z0,tPen\WObj:=wPaper;
    MoveL Offs(pOrigin,219.50,102.97,0.00),v40,z0,tPen\WObj:=wPaper;
    MoveL Offs(pOrigin,218.60,102.07,0.00),v40,z0,tPen\WObj:=wPaper;
    MoveL Offs(pOrigin,217.85,102.30,0.00),v40,z0,tPen\WObj:=wPaper;
    MoveL Offs(pOrigin,202.85,102.30,0.00),v40,fine,tPen\WObj:=wPaper;
    MoveL Offs(pOrigin,202.85,102.30,6.00),v60,z5,tPen\WObj:=wPaper;
    MoveL Offs(pOrigin,204.34,102.82,6.00),vTravel,z5,tPen\WObj:=wPaper;
    MoveL Offs(pOrigin,204.34,102.82,0.00),v60,z0,tPen\WObj:=wPaper;
    MoveL Offs(pOrigin,204.34,95.18,0.00),v40,z0,tPen\WObj:=wPaper;
    MoveL Offs(pOrigin,205.40,95.48,0.00),v40,z0,tPen\WObj:=wPaper;
    MoveL Offs(pOrigin,205.40,102.82,0.00),v40,z0,tPen\WObj:=wPaper;
    MoveL Offs(pOrigin,206.46,102.82,0.00),v40,z0,tPen\WObj:=wPaper;
    MoveL Offs(pOrigin,206.46,95.92,0.00),v40,fine,tPen\WObj:=wPaper;
    MoveL Offs(pOrigin,206.46,95.92,6.00),v60,z5,tPen\WObj:=wPaper;
    MoveL Offs(pOrigin,207.51,96.82,6.00),vTravel,z5,tPen\WObj:=wPaper;
    MoveL Offs(pOrigin,207.51,96.82,0.00),v60,z0,tPen\WObj:=wPaper;
    MoveL Offs(pOrigin,207.51,102.82,0.00),v40,z0,tPen\WObj:=wPaper;
    MoveL Offs(pOrigin,208.57,102.82,0.00),v40,z0,tPen\WObj:=wPaper;
    MoveL Offs(pOrigin,208.57,98.02,0.00),v40,fine,tPen\WObj:=wPaper;
    MoveL Offs(pOrigin,208.57,98.02,6.00),v60,z5,tPen\WObj:=wPaper;
    MoveL Offs(pOrigin,209.62,98.78,6.00),vTravel,z5,tPen\WObj:=wPaper;
    MoveL Offs(pOrigin,209.62,98.78,0.00),v60,z0,tPen\WObj:=wPaper;
    MoveL Offs(pOrigin,209.62,101.92,0.00),v40,fine,tPen\WObj:=wPaper;
    MoveL Offs(pOrigin,209.62,101.92,6.00),v60,z5,tPen\WObj:=wPaper;
    MoveL Offs(pOrigin,210.68,101.32,6.00),vTravel,z5,tPen\WObj:=wPaper;
    MoveL Offs(pOrigin,210.68,101.32,0.00),v60,z0,tPen\WObj:=wPaper;
    MoveL Offs(pOrigin,210.68,98.62,0.00),v40,fine,tPen\WObj:=wPaper;
    MoveL Offs(pOrigin,210.68,98.62,6.00),v60,z5,tPen\WObj:=wPaper;
    MoveL Offs(pOrigin,211.74,97.72,6.00),vTravel,z5,tPen\WObj:=wPaper;
    MoveL Offs(pOrigin,211.74,97.72,0.00),v60,z0,tPen\WObj:=wPaper;
    MoveL Offs(pOrigin,211.74,101.32,0.00),v40,fine,tPen\WObj:=wPaper;
    MoveL Offs(pOrigin,211.74,101.32,6.00),v60,z5,tPen\WObj:=wPaper;
    MoveL Offs(pOrigin,212.79,101.92,6.00),vTravel,z5,tPen\WObj:=wPaper;
    MoveL Offs(pOrigin,212.79,101.92,0.00),v60,z0,tPen\WObj:=wPaper;
    MoveL Offs(pOrigin,212.79,95.32,0.00),v40,z0,tPen\WObj:=wPaper;
    MoveL Offs(pOrigin,213.85,95.18,0.00),v40,z0,tPen\WObj:=wPaper;
    MoveL Offs(pOrigin,213.85,102.68,0.00),v40,z0,tPen\WObj:=wPaper;
    MoveL Offs(pOrigin,214.90,102.68,0.00),v40,z0,tPen\WObj:=wPaper;
    MoveL Offs(pOrigin,214.90,95.18,0.00),v40,z0,tPen\WObj:=wPaper;
    MoveL Offs(pOrigin,215.96,95.18,0.00),v40,z0,tPen\WObj:=wPaper;
    MoveL Offs(pOrigin,215.96,100.12,0.00),v40,fine,tPen\WObj:=wPaper;
    MoveL Offs(pOrigin,215.96,100.12,6.00),v60,z5,tPen\WObj:=wPaper;
    MoveL Offs(pOrigin,217.02,99.22,6.00),vTravel,z5,tPen\WObj:=wPaper;
    MoveL Offs(pOrigin,217.02,99.22,0.00),v60,z0,tPen\WObj:=wPaper;
    MoveL Offs(pOrigin,217.02,95.18,0.00),v40,z0,tPen\WObj:=wPaper;
    MoveL Offs(pOrigin,218.07,95.32,0.00),v40,z0,tPen\WObj:=wPaper;
    MoveL Offs(pOrigin,218.07,98.62,0.00),v40,fine,tPen\WObj:=wPaper;
    MoveL Offs(pOrigin,218.07,98.62,6.00),v60,z5,tPen\WObj:=wPaper;
    MoveL Offs(pOrigin,219.13,97.88,6.00),vTravel,z5,tPen\WObj:=wPaper;
    MoveL Offs(pOrigin,219.13,97.88,0.00),v60,z0,tPen\WObj:=wPaper;
    MoveL Offs(pOrigin,219.13,96.08,0.00),v40,fine,tPen\WObj:=wPaper;
    MoveL Offs(pOrigin,219.13,96.08,6.00),v60,z5,tPen\WObj:=wPaper;
    MoveL Offs(pOrigin,219.35,99.13,6.00),vTravel,z5,tPen\WObj:=wPaper;
    MoveL Offs(pOrigin,219.35,99.13,0.00),v60,z0,tPen\WObj:=wPaper;
    MoveL Offs(pOrigin,202.70,99.13,0.00),v40,fine,tPen\WObj:=wPaper;
    MoveL Offs(pOrigin,202.70,99.13,6.00),v60,z5,tPen\WObj:=wPaper;
    MoveL Offs(pOrigin,201.35,98.46,6.00),vTravel,z5,tPen\WObj:=wPaper;
    MoveL Offs(pOrigin,201.35,98.46,0.00),v60,z0,tPen\WObj:=wPaper;
    MoveL Offs(pOrigin,207.50,92.31,0.00),v40,z0,tPen\WObj:=wPaper;
    MoveL Offs(pOrigin,206.95,93.11,0.00),v40,z0,tPen\WObj:=wPaper;
    MoveL Offs(pOrigin,224.24,110.40,0.00),v40,fine,tPen\WObj:=wPaper;
    MoveL Offs(pOrigin,224.24,110.40,6.00),v60,z5,tPen\WObj:=wPaper;
    MoveL Offs(pOrigin,219.70,99.89,6.00),vTravel,z5,tPen\WObj:=wPaper;
    MoveL Offs(pOrigin,219.70,99.89,0.00),v60,z0,tPen\WObj:=wPaper;
    MoveL Offs(pOrigin,212.91,93.10,0.00),v40,fine,tPen\WObj:=wPaper;
    MoveL Offs(pOrigin,212.91,93.10,6.00),v60,z5,tPen\WObj:=wPaper;
    MoveL Offs(pOrigin,212.00,89.62,6.00),vTravel,z5,tPen\WObj:=wPaper;
    MoveL Offs(pOrigin,212.00,89.62,0.00),v60,z0,tPen\WObj:=wPaper;
    MoveL Offs(pOrigin,214.40,89.62,0.00),v40,fine,tPen\WObj:=wPaper;
    MoveL Offs(pOrigin,214.40,89.62,6.00),v60,z5,tPen\WObj:=wPaper;
    MoveL Offs(pOrigin,218.00,89.62,6.00),vTravel,z5,tPen\WObj:=wPaper;
    MoveL Offs(pOrigin,218.00,89.62,0.00),v60,z0,tPen\WObj:=wPaper;
    MoveL Offs(pOrigin,228.05,89.62,0.00),v40,fine,tPen\WObj:=wPaper;
    MoveL Offs(pOrigin,228.05,89.62,6.00),v60,z5,tPen\WObj:=wPaper;
    MoveL Offs(pOrigin,222.20,97.02,6.00),vTravel,z5,tPen\WObj:=wPaper;
    MoveL Offs(pOrigin,222.20,97.02,0.00),v60,z0,tPen\WObj:=wPaper;
    MoveL Offs(pOrigin,202.70,97.02,0.00),v40,fine,tPen\WObj:=wPaper;
    MoveL Offs(pOrigin,202.70,97.02,6.00),v60,z5,tPen\WObj:=wPaper;
    MoveL Offs(pOrigin,199.63,94.20,6.00),vTravel,z5,tPen\WObj:=wPaper;
    MoveL Offs(pOrigin,199.63,94.20,0.00),v60,z0,tPen\WObj:=wPaper;
    MoveL Offs(pOrigin,173.43,120.40,0.00),v40,fine,tPen\WObj:=wPaper;
    MoveL Offs(pOrigin,173.43,120.40,6.00),v60,z5,tPen\WObj:=wPaper;
    MoveL Offs(pOrigin,173.22,119.13,6.00),vTravel,z5,tPen\WObj:=wPaper;
    MoveL Offs(pOrigin,173.22,119.13,0.00),v60,z0,tPen\WObj:=wPaper;
    MoveL Offs(pOrigin,199.31,93.03,0.00),v40,z0,tPen\WObj:=wPaper;
    MoveL Offs(pOrigin,198.35,92.50,0.00),v40,z0,tPen\WObj:=wPaper;
    MoveL Offs(pOrigin,173.21,117.64,0.00),v40,fine,tPen\WObj:=wPaper;
    MoveL Offs(pOrigin,173.21,117.64,6.00),v60,z5,tPen\WObj:=wPaper;
    MoveL Offs(pOrigin,175.10,116.02,6.00),vTravel,z5,tPen\WObj:=wPaper;
    MoveL Offs(pOrigin,175.10,116.02,0.00),v60,z0,tPen\WObj:=wPaper;
    MoveL Offs(pOrigin,198.20,116.02,0.00),v40,z0,tPen\WObj:=wPaper;
    MoveL Offs(pOrigin,198.20,114.97,0.00),v40,z0,tPen\WObj:=wPaper;
    MoveL Offs(pOrigin,175.10,114.97,0.00),v40,z0,tPen\WObj:=wPaper;
    MoveL Offs(pOrigin,175.10,113.91,0.00),v40,z0,tPen\WObj:=wPaper;
    MoveL Offs(pOrigin,198.20,113.91,0.00),v40,fine,tPen\WObj:=wPaper;
  ENDPROC

  PROC DrawPart36()
    MoveL Offs(pOrigin,198.20,113.91,6.00),v60,z5,tPen\WObj:=wPaper;
    MoveL Offs(pOrigin,199.79,111.97,6.00),vTravel,z5,tPen\WObj:=wPaper;
    MoveL Offs(pOrigin,199.79,111.97,0.00),v60,z0,tPen\WObj:=wPaper;
    MoveL Offs(pOrigin,177.62,134.14,0.00),v40,fine,tPen\WObj:=wPaper;
    MoveL Offs(pOrigin,177.62,134.14,6.00),v60,z5,tPen\WObj:=wPaper;
    MoveL Offs(pOrigin,201.38,111.87,6.00),vTravel,z5,tPen\WObj:=wPaper;
    MoveL Offs(pOrigin,201.38,111.87,0.00),v60,z0,tPen\WObj:=wPaper;
    MoveL Offs(pOrigin,233.20,80.05,0.00),v40,fine,tPen\WObj:=wPaper;
    MoveL Offs(pOrigin,233.20,80.05,6.00),v60,z5,tPen\WObj:=wPaper;
    MoveL Offs(pOrigin,233.19,75.58,6.00),vTravel,z5,tPen\WObj:=wPaper;
    MoveL Offs(pOrigin,233.19,75.58,0.00),v60,z0,tPen\WObj:=wPaper;
    MoveL Offs(pOrigin,217.92,90.85,0.00),v40,fine,tPen\WObj:=wPaper;
    MoveL Offs(pOrigin,217.92,90.85,6.00),v60,z5,tPen\WObj:=wPaper;
    MoveL Offs(pOrigin,208.40,89.62,6.00),vTravel,z5,tPen\WObj:=wPaper;
    MoveL Offs(pOrigin,208.40,89.62,0.00),v60,z0,tPen\WObj:=wPaper;
    MoveL Offs(pOrigin,206.45,89.62,0.00),v40,fine,tPen\WObj:=wPaper;
    MoveL Offs(pOrigin,206.45,89.62,6.00),v60,z5,tPen\WObj:=wPaper;
    MoveL Offs(pOrigin,201.52,86.34,6.00),vTravel,z5,tPen\WObj:=wPaper;
    MoveL Offs(pOrigin,201.52,86.34,0.00),v60,z0,tPen\WObj:=wPaper;
    MoveL Offs(pOrigin,227.62,60.25,0.00),v40,fine,tPen\WObj:=wPaper;
    MoveL Offs(pOrigin,227.62,60.25,6.00),v60,z5,tPen\WObj:=wPaper;
    MoveL Offs(pOrigin,199.83,50.70,6.00),vTravel,z5,tPen\WObj:=wPaper;
    MoveL Offs(pOrigin,199.83,50.70,0.00),v60,z0,tPen\WObj:=wPaper;
    MoveL Offs(pOrigin,173.20,77.32,0.00),v40,fine,tPen\WObj:=wPaper;
    MoveL Offs(pOrigin,173.20,77.32,6.00),v60,z5,tPen\WObj:=wPaper;
    MoveL Offs(pOrigin,176.89,81.68,6.00),vTravel,z5,tPen\WObj:=wPaper;
    MoveL Offs(pOrigin,176.89,81.68,0.00),v60,z0,tPen\WObj:=wPaper;
    MoveL Offs(pOrigin,176.89,86.18,0.00),v40,fine,tPen\WObj:=wPaper;
    MoveL Offs(pOrigin,176.89,86.18,6.00),v60,z5,tPen\WObj:=wPaper;
    MoveL Offs(pOrigin,177.94,87.07,6.00),vTravel,z5,tPen\WObj:=wPaper;
    MoveL Offs(pOrigin,177.94,87.07,0.00),v60,z0,tPen\WObj:=wPaper;
    MoveL Offs(pOrigin,177.94,82.72,0.00),v40,fine,tPen\WObj:=wPaper;
    MoveL Offs(pOrigin,177.94,82.72,6.00),v60,z5,tPen\WObj:=wPaper;
    MoveL Offs(pOrigin,179.00,83.62,6.00),vTravel,z5,tPen\WObj:=wPaper;
    MoveL Offs(pOrigin,179.00,83.62,0.00),v60,z0,tPen\WObj:=wPaper;
    MoveL Offs(pOrigin,179.00,87.82,0.00),v40,z0,tPen\WObj:=wPaper;
    MoveL Offs(pOrigin,180.06,88.12,0.00),v40,z0,tPen\WObj:=wPaper;
    MoveL Offs(pOrigin,180.06,84.52,0.00),v40,fine,tPen\WObj:=wPaper;
    MoveL Offs(pOrigin,180.06,84.52,6.00),v60,z5,tPen\WObj:=wPaper;
    MoveL Offs(pOrigin,181.11,85.12,6.00),vTravel,z5,tPen\WObj:=wPaper;
    MoveL Offs(pOrigin,181.11,85.12,0.00),v60,z0,tPen\WObj:=wPaper;
    MoveL Offs(pOrigin,181.11,88.12,0.00),v40,z0,tPen\WObj:=wPaper;
    MoveL Offs(pOrigin,182.17,88.12,0.00),v40,z0,tPen\WObj:=wPaper;
    MoveL Offs(pOrigin,182.17,85.88,0.00),v40,fine,tPen\WObj:=wPaper;
    MoveL Offs(pOrigin,182.17,85.88,6.00),v60,z5,tPen\WObj:=wPaper;
    MoveL Offs(pOrigin,183.22,86.48,6.00),vTravel,z5,tPen\WObj:=wPaper;
    MoveL Offs(pOrigin,183.22,86.48,0.00),v60,z0,tPen\WObj:=wPaper;
    MoveL Offs(pOrigin,183.22,88.12,0.00),v40,fine,tPen\WObj:=wPaper;
    MoveL Offs(pOrigin,183.22,88.12,6.00),v60,z5,tPen\WObj:=wPaper;
    MoveL Offs(pOrigin,191.75,89.62,6.00),vTravel,z5,tPen\WObj:=wPaper;
    MoveL Offs(pOrigin,191.75,89.62,0.00),v60,z0,tPen\WObj:=wPaper;
    MoveL Offs(pOrigin,194.60,89.62,0.00),v40,fine,tPen\WObj:=wPaper;
    MoveL Offs(pOrigin,194.60,89.62,6.00),v60,z5,tPen\WObj:=wPaper;
    MoveL Offs(pOrigin,198.12,93.25,6.00),vTravel,z5,tPen\WObj:=wPaper;
    MoveL Offs(pOrigin,198.12,93.25,0.00),v60,z0,tPen\WObj:=wPaper;
    MoveL Offs(pOrigin,199.08,94.20,0.00),v40,z0,tPen\WObj:=wPaper;
    MoveL Offs(pOrigin,198.50,94.90,0.00),v40,z0,tPen\WObj:=wPaper;
    MoveL Offs(pOrigin,174.95,94.90,0.00),v40,z0,tPen\WObj:=wPaper;
    MoveL Offs(pOrigin,175.25,93.85,0.00),v40,z0,tPen\WObj:=wPaper;
    MoveL Offs(pOrigin,198.20,93.85,0.00),v40,fine,tPen\WObj:=wPaper;
    MoveL Offs(pOrigin,198.20,93.85,6.00),v60,z5,tPen\WObj:=wPaper;
    MoveL Offs(pOrigin,173.45,51.69,6.00),vTravel,z5,tPen\WObj:=wPaper;
    MoveL Offs(pOrigin,173.45,51.69,0.00),v60,z0,tPen\WObj:=wPaper;
    MoveL Offs(pOrigin,175.36,49.78,0.00),v40,fine,tPen\WObj:=wPaper;
    MoveL Offs(pOrigin,175.36,49.78,6.00),v60,z5,tPen\WObj:=wPaper;
    MoveL Offs(pOrigin,132.18,52.69,6.00),vTravel,z5,tPen\WObj:=wPaper;
    MoveL Offs(pOrigin,132.18,52.69,0.00),v60,z0,tPen\WObj:=wPaper;
    MoveL Offs(pOrigin,130.17,50.68,0.00),v40,fine,tPen\WObj:=wPaper;
    MoveL Offs(pOrigin,130.17,50.68,6.00),v60,z5,tPen\WObj:=wPaper;
    MoveL Offs(pOrigin,128.68,50.68,6.00),vTravel,z5,tPen\WObj:=wPaper;
    MoveL Offs(pOrigin,128.68,50.68,0.00),v60,z0,tPen\WObj:=wPaper;
    MoveL Offs(pOrigin,132.18,54.18,0.00),v40,fine,tPen\WObj:=wPaper;
    MoveL Offs(pOrigin,132.18,54.18,6.00),v60,z5,tPen\WObj:=wPaper;
    MoveL Offs(pOrigin,132.54,67.21,6.00),vTravel,z5,tPen\WObj:=wPaper;
    MoveL Offs(pOrigin,132.54,67.21,0.00),v60,z0,tPen\WObj:=wPaper;
    MoveL Offs(pOrigin,105.81,93.94,0.00),v40,fine,tPen\WObj:=wPaper;
    MoveL Offs(pOrigin,105.81,93.94,6.00),v60,z5,tPen\WObj:=wPaper;
    MoveL Offs(pOrigin,111.55,91.19,6.00),vTravel,z5,tPen\WObj:=wPaper;
    MoveL Offs(pOrigin,111.55,91.19,0.00),v60,z0,tPen\WObj:=wPaper;
    MoveL Offs(pOrigin,132.45,70.29,0.00),v40,fine,tPen\WObj:=wPaper;
    MoveL Offs(pOrigin,132.45,70.29,6.00),v60,z5,tPen\WObj:=wPaper;
    MoveL Offs(pOrigin,87.95,81.18,6.00),vTravel,z5,tPen\WObj:=wPaper;
    MoveL Offs(pOrigin,87.95,81.18,0.00),v60,z0,tPen\WObj:=wPaper;
    MoveL Offs(pOrigin,60.65,81.18,0.00),v40,fine,tPen\WObj:=wPaper;
    MoveL Offs(pOrigin,60.65,81.18,6.00),v60,z5,tPen\WObj:=wPaper;
    MoveL Offs(pOrigin,57.58,77.95,6.00),vTravel,z5,tPen\WObj:=wPaper;
    MoveL Offs(pOrigin,57.58,77.95,0.00),v60,z0,tPen\WObj:=wPaper;
    MoveL Offs(pOrigin,44.43,91.10,0.00),v40,z0,tPen\WObj:=wPaper;
    MoveL Offs(pOrigin,44.53,90.49,0.00),v40,z0,tPen\WObj:=wPaper;
    MoveL Offs(pOrigin,23.96,69.92,0.00),v40,z0,tPen\WObj:=wPaper;
    MoveL Offs(pOrigin,24.95,69.56,0.00),v40,z0,tPen\WObj:=wPaper;
    MoveL Offs(pOrigin,56.15,69.56,0.00),v40,fine,tPen\WObj:=wPaper;
    MoveL Offs(pOrigin,56.15,69.56,6.00),v60,z5,tPen\WObj:=wPaper;
    MoveL Offs(pOrigin,41.90,64.28,6.00),vTravel,z5,tPen\WObj:=wPaper;
    MoveL Offs(pOrigin,41.90,64.28,0.00),v60,z0,tPen\WObj:=wPaper;
    MoveL Offs(pOrigin,23.15,64.28,0.00),v40,fine,tPen\WObj:=wPaper;
    MoveL Offs(pOrigin,23.15,64.28,6.00),v60,z5,tPen\WObj:=wPaper;
    MoveL Offs(pOrigin,22.40,62.17,6.00),vTravel,z5,tPen\WObj:=wPaper;
    MoveL Offs(pOrigin,22.40,62.17,0.00),v60,z0,tPen\WObj:=wPaper;
    MoveL Offs(pOrigin,41.15,62.17,0.00),v40,fine,tPen\WObj:=wPaper;
    MoveL Offs(pOrigin,41.15,62.17,6.00),v60,z5,tPen\WObj:=wPaper;
    MoveL Offs(pOrigin,39.35,56.89,6.00),vTravel,z5,tPen\WObj:=wPaper;
    MoveL Offs(pOrigin,39.35,56.89,0.00),v60,z0,tPen\WObj:=wPaper;
    MoveL Offs(pOrigin,20.45,56.89,0.00),v40,fine,tPen\WObj:=wPaper;
    MoveL Offs(pOrigin,20.45,56.89,6.00),v60,z5,tPen\WObj:=wPaper;
    MoveL Offs(pOrigin,19.70,54.78,6.00),vTravel,z5,tPen\WObj:=wPaper;
    MoveL Offs(pOrigin,19.70,54.78,0.00),v60,z0,tPen\WObj:=wPaper;
    MoveL Offs(pOrigin,38.75,54.78,0.00),v40,fine,tPen\WObj:=wPaper;
    MoveL Offs(pOrigin,38.75,54.78,6.00),v60,z5,tPen\WObj:=wPaper;
    MoveL Offs(pOrigin,28.39,81.82,6.00),vTravel,z5,tPen\WObj:=wPaper;
    MoveL Offs(pOrigin,28.39,81.82,0.00),v60,z0,tPen\WObj:=wPaper;
    MoveL Offs(pOrigin,37.09,90.51,0.00),v40,z0,tPen\WObj:=wPaper;
    MoveL Offs(pOrigin,36.80,89.62,0.00),v40,z0,tPen\WObj:=wPaper;
    MoveL Offs(pOrigin,40.10,89.62,0.00),v40,fine,tPen\WObj:=wPaper;
    MoveL Offs(pOrigin,40.10,89.62,6.00),v60,z5,tPen\WObj:=wPaper;
    MoveL Offs(pOrigin,38.55,96.52,6.00),vTravel,z5,tPen\WObj:=wPaper;
    MoveL Offs(pOrigin,38.55,96.52,0.00),v60,z0,tPen\WObj:=wPaper;
    MoveL Offs(pOrigin,38.55,102.52,0.00),v40,fine,tPen\WObj:=wPaper;
    MoveL Offs(pOrigin,38.55,102.52,6.00),v60,z5,tPen\WObj:=wPaper;
    MoveL Offs(pOrigin,39.61,104.48,6.00),vTravel,z5,tPen\WObj:=wPaper;
  ENDPROC

